LIN {X 0,Y 689.264,Z 377.17,A -85,B 0,C 180,E1 32346.673,E2 32346.673} C_VEL
LIN {X 0,Y 693.662,Z 395.744,A -85,B 0,C 180,E1 32346.172,E2 32346.172} C_VEL
LIN {X 0,Y 691.445,Z 657.884,A -85,B 0,C 180,E1 32343.063,E2 32343.063} C_VEL
LIN {X 0,Y 690.51,Z 767.576,A -85,B 0,C 180,E1 32341.762,E2 32341.762} C_VEL
LIN {X 0,Y 689.952,Z 793.018,A -85,B 0,C 180,E1 32341.311,E2 32341.311} C_VEL
LIN {X 0,Y 689.325,Z 814.667,A -85,B 0,C 180,E1 32340.791,E2 32340.791} C_VEL
LIN {X 0,Y 688.609,Z 838.554,A -85,B 0,C 180,E1 32340.063,E2 32340.063} C_VEL
LIN {X 0,Y 687.794,Z 859.592,A -85,B 0,C 180,E1 32339.277,E2 32339.277} C_VEL
LIN {X 0,Y 686.919,Z 881.255,A -85,B 0,C 180,E1 32338.329,E2 32338.329} C_VEL
LIN {X 0,Y 685.951,Z 903.052,A -85,B 0,C 180,E1 32337.197,E2 32337.197} C_VEL
LIN {X 0,Y 685.057,Z 922.955,A -85,B 0,C 180,E1 32336.012,E2 32336.012} C_VEL
LIN {X 0,Y 684.091,Z 943.292,A -85,B 0,C 180,E1 32334.613,E2 32334.613} C_VEL
LIN {X 0,Y 683.28,Z 961.609,A -85,B 0,C 180,E1 32333.182,E2 32333.182} C_VEL
LIN {X 0,Y 682.482,Z 979.534,A -85,B 0,C 180,E1 32331.576,E2 32331.576} C_VEL
LIN {X 0,Y 681.841,Z 995.625,A -85,B 0,C 180,E1 32329.948,E2 32329.948} C_VEL
LIN {X 0,Y 681.258,Z 1011.229,A -85,B 0,C 180,E1 32328.129,E2 32328.129} C_VEL
LIN {X 0,Y 680.802,Z 1025.061,A -85,B 0,C 180,E1 32326.291,E2 32326.291} C_VEL
LIN {X 0,Y 680.459,Z 1037.321,A -85,B 0,C 180,E1 32324.379,E2 32324.379} C_VEL
LIN {X 0,Y 680.233,Z 1047.861,A -85,B 0,C 180,E1 32322.479,E2 32322.479} C_VEL
LIN {X 0,Y 680.077,Z 1056.896,A -85,B 0,C 180,E1 32320.504,E2 32320.504} C_VEL
LIN {X 0,Y 679.969,Z 1063.726,A -85,B 0,C 180,E1 32318.712,E2 32318.712} C_VEL
LIN {X 0,Y 679.919,Z 1070.07,A -85,B 0,C 180,E1 32316.587,E2 32316.587} C_VEL
LIN {X 0,Y 679.921,Z 1073.974,A -85,B 0,C 180,E1 32314.808,E2 32314.808} C_VEL
LIN {X 0,Y 679.908,Z 1077.017,A -85,B 0,C 180,E1 32312.782,E2 32312.782} C_VEL
LIN {X 0,Y 679.899,Z 1078.306,A -85,B 0,C 180,E1 32310.758,E2 32310.758} C_VEL
LIN {X 0,Y 679.914,Z 1078.238,A -85,B 0,C 180,E1 32308.989,E2 32308.989} C_VEL
LIN {X 0,Y 679.916,Z 1076.461,A -85,B 0,C 180,E1 32306.796,E2 32306.796} C_VEL
LIN {X 0,Y 679.923,Z 1073.496,A -85,B 0,C 180,E1 32304.938,E2 32304.938} C_VEL
LIN {X 0,Y 679.954,Z 1068.507,A -85,B 0,C 180,E1 32302.82,E2 32302.82} C_VEL
LIN {X 0,Y 679.992,Z 1062.513,A -85,B 0,C 180,E1 32300.948,E2 32300.948} C_VEL
LIN {X 0,Y 680.097,Z 1055.12,A -85,B 0,C 180,E1 32299.067,E2 32299.067} C_VEL
LIN {X 0,Y 680.283,Z 1045.255,A -85,B 0,C 180,E1 32297.031,E2 32297.031} C_VEL
LIN {X 0,Y 680.52,Z 1035.245,A -85,B 0,C 180,E1 32295.274,E2 32295.274} C_VEL
LIN {X 0,Y 680.898,Z 1021.894,A -85,B 0,C 180,E1 32293.272,E2 32293.272} C_VEL
LIN {X 0,Y 681.318,Z 1009.107,A -85,B 0,C 180,E1 32291.607,E2 32291.607} C_VEL
LIN {X 0,Y 681.951,Z 992.791,A -85,B 0,C 180,E1 32289.755,E2 32289.755} C_VEL
LIN {X 0,Y 682.561,Z 977.636,A -85,B 0,C 180,E1 32288.242,E2 32288.242} C_VEL
LIN {X 0,Y 683.397,Z 958.847,A -85,B 0,C 180,E1 32286.595,E2 32286.595} C_VEL
LIN {X 0,Y 684.206,Z 940.792,A -85,B 0,C 180,E1 32285.202,E2 32285.202} C_VEL
LIN {X 0,Y 685.184,Z 919.997,A -85,B 0,C 180,E1 32283.804,E2 32283.804} C_VEL
LIN {X 0,Y 686.049,Z 900.695,A -85,B 0,C 180,E1 32282.671,E2 32282.671} C_VEL
LIN {X 0,Y 687.089,Z 877.282,A -85,B 0,C 180,E1 32281.489,E2 32281.489} C_VEL
LIN {X 0,Y 687.891,Z 857.092,A -85,B 0,C 180,E1 32280.622,E2 32280.622} C_VEL
LIN {X 0,Y 688.774,Z 832.985,A -85,B 0,C 180,E1 32279.752,E2 32279.752} C_VEL
LIN {X 0,Y 689.455,Z 811.007,A -85,B 0,C 180,E1 32279.114,E2 32279.114} C_VEL
LIN {X 0,Y 690.143,Z 786.732,A -85,B 0,C 180,E1 32278.559,E2 32278.559} C_VEL
LIN {X 0,Y 690.547,Z 763.43,A -85,B 0,C 180,E1 32278.181,E2 32278.181} C_VEL
LIN {X 0,Y 692.558,Z 519.957,A -85,B 0,C 180,E1 32275.31,E2 32275.31} C_VEL
LIN {X 0,Y 693.501,Z 394.27,A -85,B 0,C 180,E1 32273.8,E2 32273.8} C_VEL
LIN {X 0,Y 689.198,Z 376.448,A -85,B 0,C 180,E1 32273.293,E2 32273.293} C_VEL
LIN {X 0,Y 689.442,Z 360.316,A -85,B 0,C 180,E1 32272.089,E2 32272.089} C_VEL
LIN {X 0,Y 682.414,Z 342.087,A -85,B 0,C 180,E1 32270.221,E2 32270.221} C_VEL
LIN {X 0,Y 680.484,Z 336.477,A -85,B 0,C 180,E1 32269.637,E2 32269.637} C_VEL
LIN {X 0,Y 680.477,Z 336.471,A -85,B 0,C 180,E1 32266.543,E2 32266.543} C_VEL
LIN {X 0,Y 680.457,Z 336.467,A -85,B 0,C 180,E1 32263.914,E2 32263.914} C_VEL
LIN {X 0,Y 680.531,Z 336.466,A -85,B 0,C 180,E1 32260.943,E2 32260.943} C_VEL
LIN {X 0,Y 680.456,Z 336.464,A -85,B 0,C 180,E1 32258.036,E2 32258.036} C_VEL
LIN {X 0,Y 680.505,Z 336.462,A -85,B 0,C 180,E1 32255.219,E2 32255.219} C_VEL
LIN {X 0,Y 680.464,Z 336.464,A -85,B 0,C 180,E1 32252.136,E2 32252.136} C_VEL
LIN {X 0,Y 680.466,Z 336.462,A -85,B 0,C 180,E1 32249.489,E2 32249.489} C_VEL
LIN {X 0,Y 680.505,Z 336.463,A -85,B 0,C 180,E1 32246.437,E2 32246.437} C_VEL
LIN {X 0,Y 680.455,Z 336.457,A -85,B 0,C 180,E1 32243.651,E2 32243.651} C_VEL
LIN {X 0,Y 680.524,Z 336.46,A -85,B 0,C 180,E1 32240.828,E2 32240.828} C_VEL
LIN {X 0,Y 680.464,Z 336.464,A -85,B 0,C 180,E1 32237.885,E2 32237.885} C_VEL
LIN {X 0,Y 680.467,Z 336.46,A -85,B 0,C 180,E1 32235.25,E2 32235.25} C_VEL
LIN {X 0,Y 680.508,Z 336.467,A -85,B 0,C 180,E1 32232.215,E2 32232.215} C_VEL
LIN {X 0,Y 680.457,Z 336.454,A -85,B 0,C 180,E1 32229.387,E2 32229.387} C_VEL
LIN {X 0,Y 680.531,Z 336.461,A -85,B 0,C 180,E1 32226.496,E2 32226.496} C_VEL
LIN {X 0,Y 680.46,Z 336.462,A -85,B 0,C 180,E1 32223.538,E2 32223.538} C_VEL
LIN {X 0,Y 680.482,Z 336.461,A -85,B 0,C 180,E1 32220.842,E2 32220.842} C_VEL
LIN {X 0,Y 680.477,Z 336.466,A -85,B 0,C 180,E1 32217.691,E2 32217.691} C_VEL
LIN {X 0,Y 680.461,Z 336.459,A -85,B 0,C 180,E1 32215.026,E2 32215.026} C_VEL
LIN {X 0,Y 680.525,Z 336.463,A -85,B 0,C 180,E1 32212.014,E2 32212.014} C_VEL
LIN {X 0,Y 680.457,Z 336.454,A -85,B 0,C 180,E1 32209.159,E2 32209.159} C_VEL
LIN {X 0,Y 680.516,Z 336.459,A -85,B 0,C 180,E1 32206.316,E2 32206.316} C_VEL
LIN {X 0,Y 680.47,Z 336.462,A -85,B 0,C 180,E1 32203.346,E2 32203.346} C_VEL
LIN {X 0,Y 680.473,Z 336.461,A -85,B 0,C 180,E1 32200.623,E2 32200.623} C_VEL
LIN {X 0,Y 680.501,Z 336.467,A -85,B 0,C 180,E1 32197.54,E2 32197.54} C_VEL
LIN {X 0,Y 680.458,Z 336.455,A -85,B 0,C 180,E1 32194.777,E2 32194.777} C_VEL
LIN {X 0,Y 680.532,Z 336.463,A -85,B 0,C 180,E1 32191.832,E2 32191.832} C_VEL
LIN {X 0,Y 680.52,Z 336.461,A -85,B 0,C 180,E1 32189.539,E2 32189.539} C_VEL
LIN {X 0,Y 679.466,Z 336.601,A -85,B 0,C 180,E1 32188.891,E2 32188.891} C_VEL
LIN {X 0,Y 673.041,Z 337.385,A -85,B 0,C 180,E1 32187.073,E2 32187.073} C_VEL
LIN {X 0,Y 672.523,Z 337.446,A -85,B 0,C 180,E1 32186.601,E2 32186.601} C_VEL
LIN {X 0,Y 672.587,Z 337.449,A -85,B 0,C 180,E1 32183.618,E2 32183.618} C_VEL
LIN {X 0,Y 672.523,Z 337.451,A -85,B 0,C 180,E1 32180.701,E2 32180.701} C_VEL
LIN {X 0,Y 672.573,Z 337.452,A -85,B 0,C 180,E1 32177.889,E2 32177.889} C_VEL
LIN {X 0,Y 672.529,Z 337.444,A -85,B 0,C 180,E1 32174.807,E2 32174.807} C_VEL
LIN {X 0,Y 672.538,Z 337.449,A -85,B 0,C 180,E1 32172.107,E2 32172.107} C_VEL
LIN {X 0,Y 672.553,Z 337.459,A -85,B 0,C 180,E1 32168.963,E2 32168.963} C_VEL
LIN {X 0,Y 672.551,Z 337.617,A -85,B 0,C 180,E1 32166.62,E2 32166.62} C_VEL
LIN {X 0,Y 676.581,Z 348.492,A -85,B 0,C 180,E1 32165.427,E2 32165.427} C_VEL
LIN {X 0,Y 686.819,Z 366.483,A -85,B 0,C 180,E1 32164.54,E2 32164.54} C_VEL
LIN {X 0,Y 687.145,Z 369.523,A -85,B 0,C 180,E1 32164.481,E2 32164.481} C_VEL
LIN {X 0,Y 684.937,Z 605.975,A -85,B 0,C 180,E1 32161.643,E2 32161.643} C_VEL
LIN {X 0,Y 683.701,Z 737.454,A -85,B 0,C 180,E1 32160.073,E2 32160.073} C_VEL
LIN {X 0,Y 683.098,Z 762.982,A -85,B 0,C 180,E1 32159.617,E2 32159.617} C_VEL
LIN {X 0,Y 682.418,Z 784.428,A -85,B 0,C 180,E1 32159.099,E2 32159.099} C_VEL
LIN {X 0,Y 681.594,Z 808.728,A -85,B 0,C 180,E1 32158.353,E2 32158.353} C_VEL
LIN {X 0,Y 680.746,Z 828.609,A -85,B 0,C 180,E1 32157.607,E2 32157.607} C_VEL
LIN {X 0,Y 679.837,Z 849.314,A -85,B 0,C 180,E1 32156.7,E2 32156.7} C_VEL
LIN {X 0,Y 678.703,Z 872.036,A -85,B 0,C 180,E1 32155.526,E2 32155.526} C_VEL
LIN {X 0,Y 677.739,Z 891.66,A -85,B 0,C 180,E1 32154.353,E2 32154.353} C_VEL
LIN {X 0,Y 676.632,Z 912.524,A -85,B 0,C 180,E1 32152.916,E2 32152.916} C_VEL
LIN {X 0,Y 675.764,Z 930.2,A -85,B 0,C 180,E1 32151.528,E2 32151.528} C_VEL
LIN {X 0,Y 674.826,Z 949.063,A -85,B 0,C 180,E1 32149.835,E2 32149.835} C_VEL
LIN {X 0,Y 674.128,Z 964.72,A -85,B 0,C 180,E1 32148.238,E2 32148.238} C_VEL
LIN {X 0,Y 673.443,Z 980.568,A -85,B 0,C 180,E1 32146.386,E2 32146.386} C_VEL
LIN {X 0,Y 672.97,Z 993.715,A -85,B 0,C 180,E1 32144.63,E2 32144.63} C_VEL
LIN {X 0,Y 672.58,Z 1006.12,A -85,B 0,C 180,E1 32142.71,E2 32142.71} C_VEL
LIN {X 0,Y 672.312,Z 1015.81,A -85,B 0,C 180,E1 32140.974,E2 32140.974} C_VEL
LIN {X 0,Y 672.106,Z 1025.606,A -85,B 0,C 180,E1 32138.901,E2 32138.901} C_VEL
LIN {X 0,Y 672.002,Z 1032.768,A -85,B 0,C 180,E1 32137.043,E2 32137.043} C_VEL
LIN {X 0,Y 671.953,Z 1039.052,A -85,B 0,C 180,E1 32135.037,E2 32135.037} C_VEL
LIN {X 0,Y 671.917,Z 1043.668,A -85,B 0,C 180,E1 32132.986,E2 32132.986} C_VEL
LIN {X 0,Y 671.912,Z 1046.577,A -85,B 0,C 180,E1 32131.108,E2 32131.108} C_VEL
LIN {X 0,Y 671.911,Z 1048.239,A -85,B 0,C 180,E1 32128.977,E2 32128.977} C_VEL
LIN {X 0,Y 671.901,Z 1048.306,A -85,B 0,C 180,E1 32127.185,E2 32127.185} C_VEL
LIN {X 0,Y 671.901,Z 1047.011,A -85,B 0,C 180,E1 32125.134,E2 32125.134} C_VEL
LIN {X 0,Y 671.913,Z 1044.111,A -85,B 0,C 180,E1 32123.163,E2 32123.163} C_VEL
LIN {X 0,Y 671.93,Z 1040.23,A -85,B 0,C 180,E1 32121.356,E2 32121.356} C_VEL
LIN {X 0,Y 671.979,Z 1033.919,A -85,B 0,C 180,E1 32119.194,E2 32119.194} C_VEL
LIN {X 0,Y 672.093,Z 1027.074,A -85,B 0,C 180,E1 32117.368,E2 32117.368} C_VEL
LIN {X 0,Y 672.28,Z 1018.007,A -85,B 0,C 180,E1 32115.354,E2 32115.354} C_VEL
LIN {X 0,Y 672.542,Z 1007.386,A -85,B 0,C 180,E1 32113.414,E2 32113.414} C_VEL
LIN {X 0,Y 672.926,Z 995.003,A -85,B 0,C 180,E1 32111.459,E2 32111.459} C_VEL
LIN {X 0,Y 673.43,Z 980.998,A -85,B 0,C 180,E1 32109.579,E2 32109.579} C_VEL
LIN {X 0,Y 674.098,Z 965.519,A -85,B 0,C 180,E1 32107.757,E2 32107.757} C_VEL
LIN {X 0,Y 674.815,Z 949.282,A -85,B 0,C 180,E1 32106.097,E2 32106.097} C_VEL
LIN {X 0,Y 675.726,Z 930.994,A -85,B 0,C 180,E1 32104.447,E2 32104.447} C_VEL
LIN {X 0,Y 676.583,Z 913.495,A -85,B 0,C 180,E1 32103.066,E2 32103.066} C_VEL
LIN {X 0,Y 677.683,Z 892.893,A -85,B 0,C 180,E1 32101.634,E2 32101.634} C_VEL
LIN {X 0,Y 678.634,Z 873.594,A -85,B 0,C 180,E1 32100.472,E2 32100.472} C_VEL
LIN {X 0,Y 679.741,Z 851.422,A -85,B 0,C 180,E1 32099.307,E2 32099.307} C_VEL
LIN {X 0,Y 680.676,Z 830.276,A -85,B 0,C 180,E1 32098.371,E2 32098.371} C_VEL
LIN {X 0,Y 681.516,Z 810.536,A -85,B 0,C 180,E1 32097.621,E2 32097.621} C_VEL
LIN {X 0,Y 682.396,Z 785.089,A -85,B 0,C 180,E1 32096.829,E2 32096.829} C_VEL
LIN {X 0,Y 683.074,Z 763.638,A -85,B 0,C 180,E1 32096.307,E2 32096.307} C_VEL
LIN {X 0,Y 683.695,Z 738.242,A -85,B 0,C 180,E1 32095.848,E2 32095.848} C_VEL
LIN {X 0,Y 684.492,Z 656.332,A -85,B 0,C 180,E1 32094.862,E2 32094.862} C_VEL
LIN {X 0,Y 686.784,Z 406.301,A -85,B 0,C 180,E1 32091.875,E2 32091.875} C_VEL
LIN {X 0,Y 686.991,Z 367.172,A -85,B 0,C 180,E1 32091.39,E2 32091.39} C_VEL
LIN {X 0,Y 685.188,Z 363.29,A -85,B 0,C 180,E1 32091.227,E2 32091.227} C_VEL
LIN {X 0,Y 676.327,Z 347.874,A -85,B 0,C 180,E1 32090.437,E2 32090.437} C_VEL
LIN {X 0,Y 672.529,Z 337.459,A -85,B 0,C 180,E1 32089.255,E2 32089.255} C_VEL
LIN {X 0,Y 672.582,Z 337.45,A -85,B 0,C 180,E1 32086.262,E2 32086.262} C_VEL
LIN {X 0,Y 672.521,Z 337.451,A -85,B 0,C 180,E1 32083.362,E2 32083.362} C_VEL
LIN {X 0,Y 672.589,Z 337.433,A -85,B 0,C 180,E1 32080.404,E2 32080.404} C_VEL
LIN {X 0,Y 672.522,Z 337.452,A -85,B 0,C 180,E1 32077.445,E2 32077.445} C_VEL
LIN {X 0,Y 672.565,Z 337.438,A -85,B 0,C 180,E1 32074.605,E2 32074.605} C_VEL
LIN {X 0,Y 672.531,Z 337.446,A -85,B 0,C 180,E1 32071.557,E2 32071.557} C_VEL
LIN {X 0,Y 672.53,Z 337.454,A -85,B 0,C 180,E1 32068.872,E2 32068.872} C_VEL
LIN {X 0,Y 672.568,Z 337.445,A -85,B 0,C 180,E1 32065.823,E2 32065.823} C_VEL
LIN {X 0,Y 672.52,Z 337.454,A -85,B 0,C 180,E1 32063.018,E2 32063.018} C_VEL
LIN {X 0,Y 672.592,Z 337.453,A -85,B 0,C 180,E1 32060.085,E2 32060.085} C_VEL
LIN {X 0,Y 672.52,Z 337.449,A -85,B 0,C 180,E1 32057.121,E2 32057.121} C_VEL
LIN {X 0,Y 672.551,Z 337.453,A -85,B 0,C 180,E1 32054.376,E2 32054.376} C_VEL
LIN {X 0,Y 672.532,Z 337.45,A -85,B 0,C 180,E1 32051.231,E2 32051.231} C_VEL
LIN {X 0,Y 672.528,Z 337.451,A -85,B 0,C 180,E1 32048.55,E2 32048.55} C_VEL
LIN {X 0,Y 672.576,Z 337.446,A -85,B 0,C 180,E1 32045.545,E2 32045.545} C_VEL
LIN {X 0,Y 672.517,Z 337.453,A -85,B 0,C 180,E1 32042.727,E2 32042.727} C_VEL
LIN {X 0,Y 672.59,Z 337.453,A -85,B 0,C 180,E1 32039.83,E2 32039.83} C_VEL
LIN {X 0,Y 672.522,Z 337.445,A -85,B 0,C 180,E1 32036.847,E2 32036.847} C_VEL
LIN {X 0,Y 672.542,Z 337.456,A -85,B 0,C 180,E1 32034.112,E2 32034.112} C_VEL
LIN {X 0,Y 672.534,Z 337.451,A -85,B 0,C 180,E1 32030.933,E2 32030.933} C_VEL
LIN {X 0,Y 672.522,Z 337.446,A -85,B 0,C 180,E1 32028.247,E2 32028.247} C_VEL
LIN {X 0,Y 672.586,Z 337.441,A -85,B 0,C 180,E1 32025.273,E2 32025.273} C_VEL
LIN {X 0,Y 672.517,Z 337.453,A -85,B 0,C 180,E1 32022.37,E2 32022.37} C_VEL
LIN {X 0,Y 672.585,Z 337.45,A -85,B 0,C 180,E1 32019.461,E2 32019.461} C_VEL
LIN {X 0,Y 672.521,Z 337.445,A -85,B 0,C 180,E1 32016.518,E2 32016.518} C_VEL
LIN {X 0,Y 672.539,Z 337.455,A -85,B 0,C 180,E1 32013.796,E2 32013.796} C_VEL
LIN {X 0,Y 672.535,Z 337.45,A -85,B 0,C 180,E1 32010.602,E2 32010.602} C_VEL
LIN {X 0,Y 672.521,Z 337.455,A -85,B 0,C 180,E1 32007.937,E2 32007.937} C_VEL
LIN {X 0,Y 672.584,Z 337.452,A -85,B 0,C 180,E1 32004.981,E2 32004.981} C_VEL
LIN {X 0,Y 672.517,Z 337.453,A -85,B 0,C 180,E1 32002.117,E2 32002.117} C_VEL
LIN {X 0,Y 672.567,Z 337.455,A -85,B 0,C 180,E1 31999.306,E2 31999.306} C_VEL
LIN {X 0,Y 672.526,Z 337.453,A -85,B 0,C 180,E1 31996.263,E2 31996.263} C_VEL
LIN {X 0,Y 672.526,Z 337.458,A -85,B 0,C 180,E1 31993.609,E2 31993.609} C_VEL
LIN {X 0,Y 672.592,Z 337.467,A -85,B 0,C 180,E1 31990.826,E2 31990.826} C_VEL
LIN {X 0,Y 682.601,Z 364.163,A -85,B 0,C 180,E1 31988.045,E2 31988.045} C_VEL
LIN {X 0,Y 682.307,Z 376.941,A -85,B 0,C 180,E1 31987.109,E2 31987.109} C_VEL
LIN {X 0,Y 687.167,Z 397.582,A -85,B 0,C 180,E1 31986.542,E2 31986.542} C_VEL
LIN {X 0,Y 684.716,Z 660.338,A -85,B 0,C 180,E1 31983.4,E2 31983.4} C_VEL
LIN {X 0,Y 683.699,Z 767.71,A -85,B 0,C 180,E1 31982.114,E2 31982.114} C_VEL
LIN {X 0,Y 683.091,Z 793.146,A -85,B 0,C 180,E1 31981.658,E2 31981.658} C_VEL
LIN {X 0,Y 682.412,Z 814.556,A -85,B 0,C 180,E1 31981.14,E2 31981.14} C_VEL
LIN {X 0,Y 681.585,Z 838.968,A -85,B 0,C 180,E1 31980.39,E2 31980.39} C_VEL
LIN {X 0,Y 680.717,Z 859.347,A -85,B 0,C 180,E1 31979.622,E2 31979.622} C_VEL
LIN {X 0,Y 679.794,Z 880.266,A -85,B 0,C 180,E1 31978.701,E2 31978.701} C_VEL
LIN {X 0,Y 678.692,Z 902.317,A -85,B 0,C 180,E1 31977.555,E2 31977.555} C_VEL
LIN {X 0,Y 677.757,Z 921.216,A -85,B 0,C 180,E1 31976.426,E2 31976.426} C_VEL
LIN {X 0,Y 676.663,Z 942.008,A -85,B 0,C 180,E1 31975,E2 31975} C_VEL
LIN {X 0,Y 675.802,Z 959.4,A -85,B 0,C 180,E1 31973.638,E2 31973.638} C_VEL
LIN {X 0,Y 674.844,Z 978.606,A -85,B 0,C 180,E1 31971.924,E2 31971.924} C_VEL
LIN {X 0,Y 674.17,Z 993.722,A -85,B 0,C 180,E1 31970.389,E2 31970.389} C_VEL
LIN {X 0,Y 673.468,Z 1009.816,A -85,B 0,C 180,E1 31968.525,E2 31968.525} C_VEL
LIN {X 0,Y 673.008,Z 1022.525,A -85,B 0,C 180,E1 31966.841,E2 31966.841} C_VEL
LIN {X 0,Y 672.584,Z 1035.764,A -85,B 0,C 180,E1 31964.815,E2 31964.815} C_VEL
LIN {X 0,Y 672.325,Z 1045.586,A -85,B 0,C 180,E1 31963.061,E2 31963.061} C_VEL
LIN {X 0,Y 672.117,Z 1055.476,A -85,B 0,C 180,E1 31960.977,E2 31960.977} C_VEL
LIN {X 0,Y 672.012,Z 1062.514,A -85,B 0,C 180,E1 31959.161,E2 31959.161} C_VEL
LIN {X 0,Y 671.958,Z 1068.761,A -85,B 0,C 180,E1 31957.18,E2 31957.18} C_VEL
LIN {X 0,Y 671.924,Z 1073.497,A -85,B 0,C 180,E1 31955.123,E2 31955.123} C_VEL
LIN {X 0,Y 671.916,Z 1076.462,A -85,B 0,C 180,E1 31953.242,E2 31953.242} C_VEL
LIN {X 0,Y 671.914,Z 1078.238,A -85,B 0,C 180,E1 31951.023,E2 31951.023} C_VEL
LIN {X 0,Y 671.899,Z 1078.306,A -85,B 0,C 180,E1 31949.233,E2 31949.233} C_VEL
LIN {X 0,Y 671.909,Z 1077.017,A -85,B 0,C 180,E1 31947.185,E2 31947.185} C_VEL
LIN {X 0,Y 671.922,Z 1073.974,A -85,B 0,C 180,E1 31945.134,E2 31945.134} C_VEL
LIN {X 0,Y 671.923,Z 1070.07,A -85,B 0,C 180,E1 31943.335,E2 31943.335} C_VEL
LIN {X 0,Y 671.979,Z 1063.726,A -85,B 0,C 180,E1 31941.184,E2 31941.184} C_VEL
LIN {X 0,Y 672.097,Z 1056.896,A -85,B 0,C 180,E1 31939.369,E2 31939.369} C_VEL
LIN {X 0,Y 672.282,Z 1047.686,A -85,B 0,C 180,E1 31937.338,E2 31937.338} C_VEL
LIN {X 0,Y 672.539,Z 1037.261,A -85,B 0,C 180,E1 31935.437,E2 31935.437} C_VEL
LIN {X 0,Y 672.919,Z 1025.063,A -85,B 0,C 180,E1 31933.512,E2 31933.512} C_VEL
LIN {X 0,Y 673.423,Z 1011.227,A -85,B 0,C 180,E1 31931.653,E2 31931.653} C_VEL
LIN {X 0,Y 674.071,Z 996.17,A -85,B 0,C 180,E1 31929.871,E2 31929.871} C_VEL
LIN {X 0,Y 674.76,Z 980.459,A -85,B 0,C 180,E1 31928.256,E2 31928.256} C_VEL
LIN {X 0,Y 675.65,Z 962.715,A -85,B 0,C 180,E1 31926.634,E2 31926.634} C_VEL
LIN {X 0,Y 676.557,Z 944.067,A -85,B 0,C 180,E1 31925.154,E2 31925.154} C_VEL
LIN {X 0,Y 677.598,Z 924.668,A -85,B 0,C 180,E1 31923.792,E2 31923.792} C_VEL
LIN {X 0,Y 678.618,Z 903.936,A -85,B 0,C 180,E1 31922.537,E2 31922.537} C_VEL
LIN {X 0,Y 679.681,Z 882.64,A -85,B 0,C 180,E1 31921.41,E2 31921.41} C_VEL
LIN {X 0,Y 680.68,Z 860.265,A -85,B 0,C 180,E1 31920.415,E2 31920.415} C_VEL
LIN {X 0,Y 681.547,Z 839.834,A -85,B 0,C 180,E1 31919.641,E2 31919.641} C_VEL
LIN {X 0,Y 682.405,Z 814.776,A -85,B 0,C 180,E1 31918.866,E2 31918.866} C_VEL
LIN {X 0,Y 683.086,Z 793.282,A -85,B 0,C 180,E1 31918.344,E2 31918.344} C_VEL
LIN {X 0,Y 683.699,Z 767.822,A -85,B 0,C 180,E1 31917.887,E2 31917.887} C_VEL
LIN {X 0,Y 684.658,Z 666.935,A -85,B 0,C 180,E1 31916.678,E2 31916.678} C_VEL
LIN {X 0,Y 687.132,Z 401.239,A -85,B 0,C 180,E1 31913.502,E2 31913.502} C_VEL
LIN {X 0,Y 686.935,Z 395.795,A -85,B 0,C 180,E1 31913.42,E2 31913.42} C_VEL
LIN {X 0,Y 682.24,Z 376.221,A -85,B 0,C 180,E1 31912.856,E2 31912.856} C_VEL
LIN {X 0,Y 682.47,Z 363.779,A -85,B 0,C 180,E1 31911.917,E2 31911.917} C_VEL
LIN {X 0,Y 674.923,Z 343.947,A -85,B 0,C 180,E1 31909.858,E2 31909.858} C_VEL
LIN {X 0,Y 672.591,Z 337.458,A -85,B 0,C 180,E1 31909.148,E2 31909.148} C_VEL
LIN {X 0,Y 672.521,Z 337.459,A -85,B 0,C 180,E1 31906.263,E2 31906.263} C_VEL
LIN {X 0,Y 672.537,Z 337.455,A -85,B 0,C 180,E1 31903.611,E2 31903.611} C_VEL
LIN {X 0,Y 672.535,Z 337.451,A -85,B 0,C 180,E1 31900.408,E2 31900.408} C_VEL
LIN {X 0,Y 672.521,Z 337.451,A -85,B 0,C 180,E1 31897.724,E2 31897.724} C_VEL
LIN {X 0,Y 672.58,Z 337.449,A -85,B 0,C 180,E1 31894.703,E2 31894.703} C_VEL
LIN {X 0,Y 672.515,Z 337.451,A -85,B 0,C 180,E1 31891.858,E2 31891.858} C_VEL
LIN {X 0,Y 672.574,Z 337.449,A -85,B 0,C 180,E1 31889.055,E2 31889.055} C_VEL
LIN {X 0,Y 672.526,Z 337.454,A -85,B 0,C 180,E1 31886.015,E2 31886.015} C_VEL
LIN {X 0,Y 672.535,Z 337.443,A -85,B 0,C 180,E1 31883.296,E2 31883.296} C_VEL
LIN {X 0,Y 672.538,Z 337.449,A -85,B 0,C 180,E1 31880.087,E2 31880.087} C_VEL
LIN {X 0,Y 672.525,Z 337.451,A -85,B 0,C 180,E1 31877.349,E2 31877.349} C_VEL
LIN {X 0,Y 672.574,Z 337.446,A -85,B 0,C 180,E1 31874.287,E2 31874.287} C_VEL
LIN {X 0,Y 672.518,Z 337.452,A -85,B 0,C 180,E1 31871.492,E2 31871.492} C_VEL
LIN {X 0,Y 672.582,Z 337.44,A -85,B 0,C 180,E1 31868.636,E2 31868.636} C_VEL
LIN {X 0,Y 672.525,Z 337.449,A -85,B 0,C 180,E1 31865.631,E2 31865.631} C_VEL
LIN {X 0,Y 672.541,Z 337.447,A -85,B 0,C 180,E1 31862.897,E2 31862.897} C_VEL
LIN {X 0,Y 672.538,Z 337.444,A -85,B 0,C 180,E1 31859.744,E2 31859.744} C_VEL
LIN {X 0,Y 672.525,Z 337.451,A -85,B 0,C 180,E1 31857.017,E2 31857.017} C_VEL
LIN {X 0,Y 672.583,Z 337.444,A -85,B 0,C 180,E1 31854.022,E2 31854.022} C_VEL
LIN {X 0,Y 672.519,Z 337.453,A -85,B 0,C 180,E1 31851.191,E2 31851.191} C_VEL
LIN {X 0,Y 672.576,Z 337.439,A -85,B 0,C 180,E1 31848.335,E2 31848.335} C_VEL
LIN {X 0,Y 672.529,Z 337.451,A -85,B 0,C 180,E1 31845.36,E2 31845.36} C_VEL
LIN {X 0,Y 672.537,Z 337.447,A -85,B 0,C 180,E1 31842.612,E2 31842.612} C_VEL
LIN {X 0,Y 672.546,Z 337.446,A -85,B 0,C 180,E1 31839.46,E2 31839.46} C_VEL
LIN {X 0,Y 672.527,Z 337.452,A -85,B 0,C 180,E1 31836.704,E2 31836.704} C_VEL
LIN {X 0,Y 672.585,Z 337.446,A -85,B 0,C 180,E1 31833.694,E2 31833.694} C_VEL
LIN {X 0,Y 672.522,Z 337.445,A -85,B 0,C 180,E1 31830.813,E2 31830.813} C_VEL
LIN {X 0,Y 672.585,Z 337.45,A -85,B 0,C 180,E1 31827.928,E2 31827.928} C_VEL
LIN {X 0,Y 672.523,Z 337.446,A -85,B 0,C 180,E1 31826.601,E2 31826.601} C_VEL
LIN {X 0,Y 671.558,Z 337.57,A -85,B 0,C 180,E1 31825.945,E2 31825.945} C_VEL
LIN {X 0,Y 665.187,Z 338.373,A -85,B 0,C 180,E1 31824.105,E2 31824.105} C_VEL
LIN {X 0,Y 664.648,Z 338.437,A -85,B 0,C 180,E1 31823.627,E2 31823.627} C_VEL
LIN {X 0,Y 664.585,Z 338.44,A -85,B 0,C 180,E1 31820.698,E2 31820.698} C_VEL
LIN {X 0,Y 664.638,Z 338.441,A -85,B 0,C 180,E1 31817.858,E2 31817.858} C_VEL
LIN {X 0,Y 664.596,Z 338.429,A -85,B 0,C 180,E1 31814.877,E2 31814.877} C_VEL
LIN {X 0,Y 664.598,Z 338.439,A -85,B 0,C 180,E1 31812.121,E2 31812.121} C_VEL
LIN {X 0,Y 664.611,Z 338.448,A -85,B 0,C 180,E1 31808.939,E2 31808.939} C_VEL
LIN {X 0,Y 664.652,Z 338.576,A -85,B 0,C 180,E1 31807.103,E2 31807.103} C_VEL
LIN {X 0,Y 668.468,Z 348.792,A -85,B 0,C 180,E1 31805.961,E2 31805.961} C_VEL
LIN {X 0,Y 680.723,Z 370.08,A -85,B 0,C 180,E1 31804.878,E2 31804.878} C_VEL
LIN {X 0,Y 678.272,Z 606.578,A -85,B 0,C 180,E1 31802.012,E2 31802.012} C_VEL
LIN {X 0,Y 676.917,Z 737.51,A -85,B 0,C 180,E1 31800.433,E2 31800.433} C_VEL
LIN {X 0,Y 676.265,Z 763.04,A -85,B 0,C 180,E1 31799.973,E2 31799.973} C_VEL
LIN {X 0,Y 675.538,Z 784.266,A -85,B 0,C 180,E1 31799.456,E2 31799.456} C_VEL
LIN {X 0,Y 674.669,Z 807.51,A -85,B 0,C 180,E1 31798.746,E2 31798.746} C_VEL
LIN {X 0,Y 673.656,Z 829.251,A -85,B 0,C 180,E1 31797.923,E2 31797.923} C_VEL
LIN {X 0,Y 672.621,Z 850.868,A -85,B 0,C 180,E1 31796.962,E2 31796.962} C_VEL
LIN {X 0,Y 671.416,Z 872.5,A -85,B 0,C 180,E1 31795.823,E2 31795.823} C_VEL
LIN {X 0,Y 670.363,Z 892.083,A -85,B 0,C 180,E1 31794.639,E2 31794.639} C_VEL
LIN {X 0,Y 669.153,Z 912.814,A -85,B 0,C 180,E1 31793.192,E2 31793.192} C_VEL
LIN {X 0,Y 668.189,Z 930.522,A -85,B 0,C 180,E1 31791.784,E2 31791.784} C_VEL
LIN {X 0,Y 667.206,Z 948.416,A -85,B 0,C 180,E1 31790.162,E2 31790.162} C_VEL
LIN {X 0,Y 666.442,Z 963.293,A -85,B 0,C 180,E1 31788.637,E2 31788.637} C_VEL
LIN {X 0,Y 665.641,Z 980.076,A -85,B 0,C 180,E1 31786.673,E2 31786.673} C_VEL
LIN {X 0,Y 665.148,Z 992.639,A -85,B 0,C 180,E1 31784.985,E2 31784.985} C_VEL
LIN {X 0,Y 664.658,Z 1006.176,A -85,B 0,C 180,E1 31782.881,E2 31782.881} C_VEL
LIN {X 0,Y 664.357,Z 1015.988,A -85,B 0,C 180,E1 31781.098,E2 31781.098} C_VEL
LIN {X 0,Y 664.129,Z 1025.709,A -85,B 0,C 180,E1 31779.008,E2 31779.008} C_VEL
LIN {X 0,Y 664.025,Z 1032.677,A -85,B 0,C 180,E1 31777.18,E2 31777.18} C_VEL
LIN {X 0,Y 663.955,Z 1038.873,A -85,B 0,C 180,E1 31775.184,E2 31775.184} C_VEL
LIN {X 0,Y 663.92,Z 1043.554,A -85,B 0,C 180,E1 31773.108,E2 31773.108} C_VEL
LIN {X 0,Y 663.911,Z 1046.385,A -85,B 0,C 180,E1 31771.294,E2 31771.294} C_VEL
LIN {X 0,Y 663.912,Z 1048.199,A -85,B 0,C 180,E1 31769.137,E2 31769.137} C_VEL
LIN {X 0,Y 663.899,Z 1048.322,A -85,B 0,C 180,E1 31767.238,E2 31767.238} C_VEL
LIN {X 0,Y 663.898,Z 1047.134,A -85,B 0,C 180,E1 31765.248,E2 31765.248} C_VEL
LIN {X 0,Y 663.913,Z 1044.224,A -85,B 0,C 180,E1 31763.167,E2 31763.167} C_VEL
LIN {X 0,Y 663.933,Z 1040.377,A -85,B 0,C 180,E1 31761.338,E2 31761.338} C_VEL
LIN {X 0,Y 663.986,Z 1034.441,A -85,B 0,C 180,E1 31759.238,E2 31759.238} C_VEL
LIN {X 0,Y 664.109,Z 1027.328,A -85,B 0,C 180,E1 31757.302,E2 31757.302} C_VEL
LIN {X 0,Y 664.305,Z 1018.729,A -85,B 0,C 180,E1 31755.353,E2 31755.353} C_VEL
LIN {X 0,Y 664.592,Z 1008.272,A -85,B 0,C 180,E1 31753.39,E2 31753.39} C_VEL
LIN {X 0,Y 664.959,Z 997.182,A -85,B 0,C 180,E1 31751.592,E2 31751.592} C_VEL
LIN {X 0,Y 665.538,Z 982.914,A -85,B 0,C 180,E1 31749.601,E2 31749.601} C_VEL
LIN {X 0,Y 666.139,Z 969.457,A -85,B 0,C 180,E1 31747.96,E2 31747.96} C_VEL
LIN {X 0,Y 667.005,Z 952.253,A -85,B 0,C 180,E1 31746.125,E2 31746.125} C_VEL
LIN {X 0,Y 667.84,Z 936.516,A -85,B 0,C 180,E1 31744.647,E2 31744.647} C_VEL
LIN {X 0,Y 668.968,Z 916.216,A -85,B 0,C 180,E1 31742.975,E2 31742.975} C_VEL
LIN {X 0,Y 670.033,Z 897.67,A -85,B 0,C 180,E1 31741.641,E2 31741.641} C_VEL
LIN {X 0,Y 671.267,Z 875.582,A -85,B 0,C 180,E1 31740.263,E2 31740.263} C_VEL
LIN {X 0,Y 672.336,Z 855.537,A -85,B 0,C 180,E1 31739.18,E2 31739.18} C_VEL
LIN {X 0,Y 673.539,Z 831.903,A -85,B 0,C 180,E1 31738.096,E2 31738.096} C_VEL
LIN {X 0,Y 674.443,Z 812.39,A -85,B 0,C 180,E1 31737.341,E2 31737.341} C_VEL
LIN {X 0,Y 675.396,Z 788.595,A -85,B 0,C 180,E1 31736.57,E2 31736.57} C_VEL
LIN {X 0,Y 676.156,Z 765.864,A -85,B 0,C 180,E1 31735.999,E2 31735.999} C_VEL
LIN {X 0,Y 676.874,Z 741.591,A -85,B 0,C 180,E1 31735.535,E2 31735.535} C_VEL
LIN {X 0,Y 677.412,Z 695.138,A -85,B 0,C 180,E1 31734.953,E2 31734.953} C_VEL
LIN {X 0,Y 679.97,Z 442.631,A -85,B 0,C 180,E1 31731.92,E2 31731.92} C_VEL
LIN {X 0,Y 680.612,Z 369.671,A -85,B 0,C 180,E1 31731.02,E2 31731.02} C_VEL
LIN {X 0,Y 668.308,Z 348.44,A -85,B 0,C 180,E1 31729.932,E2 31729.932} C_VEL
LIN {X 0,Y 664.639,Z 338.439,A -85,B 0,C 180,E1 31728.782,E2 31728.782} C_VEL
LIN {X 0,Y 664.589,Z 338.441,A -85,B 0,C 180,E1 31725.725,E2 31725.725} C_VEL
LIN {X 0,Y 664.604,Z 338.442,A -85,B 0,C 180,E1 31722.964,E2 31722.964} C_VEL
LIN {X 0,Y 664.597,Z 338.435,A -85,B 0,C 180,E1 31719.748,E2 31719.748} C_VEL
LIN {X 0,Y 664.593,Z 338.44,A -85,B 0,C 180,E1 31717,E2 31717} C_VEL
LIN {X 0,Y 664.619,Z 338.439,A -85,B 0,C 180,E1 31713.854,E2 31713.854} C_VEL
LIN {X 0,Y 664.585,Z 338.437,A -85,B 0,C 180,E1 31711.068,E2 31711.068} C_VEL
LIN {X 0,Y 664.653,Z 338.437,A -85,B 0,C 180,E1 31708.091,E2 31708.091} C_VEL
LIN {X 0,Y 664.58,Z 338.436,A -85,B 0,C 180,E1 31705.201,E2 31705.201} C_VEL
LIN {X 0,Y 664.631,Z 338.441,A -85,B 0,C 180,E1 31702.372,E2 31702.372} C_VEL
LIN {X 0,Y 664.592,Z 338.44,A -85,B 0,C 180,E1 31699.329,E2 31699.329} C_VEL
LIN {X 0,Y 664.597,Z 338.441,A -85,B 0,C 180,E1 31696.59,E2 31696.59} C_VEL
LIN {X 0,Y 664.604,Z 338.437,A -85,B 0,C 180,E1 31693.397,E2 31693.397} C_VEL
LIN {X 0,Y 664.584,Z 338.442,A -85,B 0,C 180,E1 31690.665,E2 31690.665} C_VEL
LIN {X 0,Y 664.645,Z 338.437,A -85,B 0,C 180,E1 31687.608,E2 31687.608} C_VEL
LIN {X 0,Y 664.579,Z 338.438,A -85,B 0,C 180,E1 31684.747,E2 31684.747} C_VEL
LIN {X 0,Y 664.647,Z 338.434,A -85,B 0,C 180,E1 31681.81,E2 31681.81} C_VEL
LIN {X 0,Y 664.585,Z 338.441,A -85,B 0,C 180,E1 31678.879,E2 31678.879} C_VEL
LIN {X 0,Y 664.606,Z 338.437,A -85,B 0,C 180,E1 31676.118,E2 31676.118} C_VEL
LIN {X 0,Y 664.596,Z 338.431,A -85,B 0,C 180,E1 31673,E2 31673} C_VEL
LIN {X 0,Y 664.584,Z 338.443,A -85,B 0,C 180,E1 31670.299,E2 31670.299} C_VEL
LIN {X 0,Y 664.636,Z 338.438,A -85,B 0,C 180,E1 31667.223,E2 31667.223} C_VEL
LIN {X 0,Y 664.578,Z 338.434,A -85,B 0,C 180,E1 31664.376,E2 31664.376} C_VEL
LIN {X 0,Y 664.651,Z 338.433,A -85,B 0,C 180,E1 31661.402,E2 31661.402} C_VEL
LIN {X 0,Y 664.58,Z 338.442,A -85,B 0,C 180,E1 31658.405,E2 31658.405} C_VEL
LIN {X 0,Y 664.631,Z 338.438,A -85,B 0,C 180,E1 31655.561,E2 31655.561} C_VEL
LIN {X 0,Y 664.587,Z 338.437,A -85,B 0,C 180,E1 31652.491,E2 31652.491} C_VEL
LIN {X 0,Y 664.591,Z 338.443,A -85,B 0,C 180,E1 31649.834,E2 31649.834} C_VEL
LIN {X 0,Y 664.613,Z 338.441,A -85,B 0,C 180,E1 31646.692,E2 31646.692} C_VEL
LIN {X 0,Y 664.58,Z 338.444,A -85,B 0,C 180,E1 31643.965,E2 31643.965} C_VEL
LIN {X 0,Y 664.653,Z 338.44,A -85,B 0,C 180,E1 31641.036,E2 31641.036} C_VEL
LIN {X 0,Y 664.579,Z 338.443,A -85,B 0,C 180,E1 31638.085,E2 31638.085} C_VEL
LIN {X 0,Y 664.627,Z 338.442,A -85,B 0,C 180,E1 31635.243,E2 31635.243} C_VEL
LIN {X 0,Y 664.585,Z 338.443,A -85,B 0,C 180,E1 31632.146,E2 31632.146} C_VEL
LIN {X 0,Y 664.621,Z 338.542,A -85,B 0,C 180,E1 31631.317,E2 31631.317} C_VEL
LIN {X 0,Y 673.506,Z 362.08,A -85,B 0,C 180,E1 31628.792,E2 31628.792} C_VEL
LIN {X 0,Y 675.561,Z 368.02,A -85,B 0,C 180,E1 31628.193,E2 31628.193} C_VEL
LIN {X 0,Y 675.363,Z 376.661,A -85,B 0,C 180,E1 31627.557,E2 31627.557} C_VEL
LIN {X 0,Y 680.703,Z 399.355,A -85,B 0,C 180,E1 31626.921,E2 31626.921} C_VEL
LIN {X 0,Y 678.008,Z 663.113,A -85,B 0,C 180,E1 31623.74,E2 31623.74} C_VEL
LIN {X 0,Y 676.914,Z 767.818,A -85,B 0,C 180,E1 31622.474,E2 31622.474} C_VEL
LIN {X 0,Y 676.255,Z 793.274,A -85,B 0,C 180,E1 31622.013,E2 31622.013} C_VEL
LIN {X 0,Y 675.528,Z 814.444,A -85,B 0,C 180,E1 31621.497,E2 31621.497} C_VEL
LIN {X 0,Y 674.622,Z 838.547,A -85,B 0,C 180,E1 31620.753,E2 31620.753} C_VEL
LIN {X 0,Y 673.655,Z 859.342,A -85,B 0,C 180,E1 31619.964,E2 31619.964} C_VEL
LIN {X 0,Y 672.656,Z 880.17,A -85,B 0,C 180,E1 31619.039,E2 31619.039} C_VEL
LIN {X 0,Y 671.429,Z 902.313,A -85,B 0,C 180,E1 31617.879,E2 31617.879} C_VEL
LIN {X 0,Y 670.354,Z 922.188,A -85,B 0,C 180,E1 31616.677,E2 31616.677} C_VEL
LIN {X 0,Y 669.167,Z 942.614,A -85,B 0,C 180,E1 31615.252,E2 31615.252} C_VEL
LIN {X 0,Y 668.229,Z 959.683,A -85,B 0,C 180,E1 31613.899,E2 31613.899} C_VEL
LIN {X 0,Y 667.192,Z 978.606,A -85,B 0,C 180,E1 31612.189,E2 31612.189} C_VEL
LIN {X 0,Y 666.433,Z 993.633,A -85,B 0,C 180,E1 31610.645,E2 31610.645} C_VEL
LIN {X 0,Y 665.654,Z 1009.818,A -85,B 0,C 180,E1 31608.751,E2 31608.751} C_VEL
LIN {X 0,Y 665.145,Z 1022.539,A -85,B 0,C 180,E1 31607.044,E2 31607.044} C_VEL
LIN {X 0,Y 664.665,Z 1035.765,A -85,B 0,C 180,E1 31604.996,E2 31604.996} C_VEL
LIN {X 0,Y 664.369,Z 1045.92,A -85,B 0,C 180,E1 31603.156,E2 31603.156} C_VEL
LIN {X 0,Y 664.133,Z 1055.927,A -85,B 0,C 180,E1 31601,E2 31601} C_VEL
LIN {X 0,Y 664.022,Z 1062.817,A -85,B 0,C 180,E1 31599.185,E2 31599.185} C_VEL
LIN {X 0,Y 663.962,Z 1069.244,A -85,B 0,C 180,E1 31597.093,E2 31597.093} C_VEL
LIN {X 0,Y 663.925,Z 1073.656,A -85,B 0,C 180,E1 31595.098,E2 31595.098} C_VEL
LIN {X 0,Y 663.917,Z 1076.574,A -85,B 0,C 180,E1 31593.194,E2 31593.194} C_VEL
LIN {X 0,Y 663.91,Z 1078.261,A -85,B 0,C 180,E1 31590.949,E2 31590.949} C_VEL
LIN {X 0,Y 663.905,Z 1078.283,A -85,B 0,C 180,E1 31589.137,E2 31589.137} C_VEL
LIN {X 0,Y 663.916,Z 1076.799,A -85,B 0,C 180,E1 31586.978,E2 31586.978} C_VEL
LIN {X 0,Y 663.925,Z 1073.815,A -85,B 0,C 180,E1 31584.989,E2 31584.989} C_VEL
LIN {X 0,Y 663.956,Z 1069.451,A -85,B 0,C 180,E1 31582.993,E2 31582.993} C_VEL
LIN {X 0,Y 664.011,Z 1063.119,A -85,B 0,C 180,E1 31580.903,E2 31580.903} C_VEL
LIN {X 0,Y 664.128,Z 1056.186,A -85,B 0,C 180,E1 31579.065,E2 31579.065} C_VEL
LIN {X 0,Y 664.356,Z 1046.484,A -85,B 0,C 180,E1 31576.953,E2 31576.953} C_VEL
LIN {X 0,Y 664.649,Z 1036.288,A -85,B 0,C 180,E1 31575.093,E2 31575.093} C_VEL
LIN {X 0,Y 665.121,Z 1023.16,A -85,B 0,C 180,E1 31573.044,E2 31573.044} C_VEL
LIN {X 0,Y 665.624,Z 1010.525,A -85,B 0,C 180,E1 31571.339,E2 31571.339} C_VEL
LIN {X 0,Y 666.404,Z 994.378,A -85,B 0,C 180,E1 31569.435,E2 31569.435} C_VEL
LIN {X 0,Y 667.168,Z 979.013,A -85,B 0,C 180,E1 31567.851,E2 31567.851} C_VEL
LIN {X 0,Y 668.189,Z 960.506,A -85,B 0,C 180,E1 31566.17,E2 31566.17} C_VEL
LIN {X 0,Y 669.129,Z 943.22,A -85,B 0,C 180,E1 31564.794,E2 31564.794} C_VEL
LIN {X 0,Y 670.317,Z 922.909,A -85,B 0,C 180,E1 31563.369,E2 31563.369} C_VEL
LIN {X 0,Y 671.389,Z 903.048,A -85,B 0,C 180,E1 31562.163,E2 31562.163} C_VEL
LIN {X 0,Y 672.604,Z 881.268,A -85,B 0,C 180,E1 31561.012,E2 31561.012} C_VEL
LIN {X 0,Y 673.605,Z 860.476,A -85,B 0,C 180,E1 31560.082,E2 31560.082} C_VEL
LIN {X 0,Y 674.538,Z 840.351,A -85,B 0,C 180,E1 31559.312,E2 31559.312} C_VEL
LIN {X 0,Y 675.503,Z 815.099,A -85,B 0,C 180,E1 31558.521,E2 31558.521} C_VEL
LIN {X 0,Y 676.235,Z 793.801,A -85,B 0,C 180,E1 31557.998,E2 31557.998} C_VEL
LIN {X 0,Y 676.909,Z 768.357,A -85,B 0,C 180,E1 31557.534,E2 31557.534} C_VEL
LIN {X 0,Y 677.778,Z 687.025,A -85,B 0,C 180,E1 31556.545,E2 31556.545} C_VEL
LIN {X 0,Y 680.316,Z 433.987,A -85,B 0,C 180,E1 31553.5,E2 31553.5} C_VEL
LIN {X 0,Y 680.519,Z 397.746,A -85,B 0,C 180,E1 31553.046,E2 31553.046} C_VEL
LIN {X 0,Y 675.309,Z 375.991,A -85,B 0,C 180,E1 31552.409,E2 31552.409} C_VEL
LIN {X 0,Y 675.511,Z 367.275,A -85,B 0,C 180,E1 31551.744,E2 31551.744} C_VEL
LIN {X 0,Y 667.62,Z 346.692,A -85,B 0,C 180,E1 31549.571,E2 31549.571} C_VEL
LIN {X 0,Y 664.607,Z 338.449,A -85,B 0,C 180,E1 31548.655,E2 31548.655} C_VEL
LIN {X 0,Y 664.579,Z 338.447,A -85,B 0,C 180,E1 31545.965,E2 31545.965} C_VEL
LIN {X 0,Y 664.647,Z 338.444,A -85,B 0,C 180,E1 31542.96,E2 31542.96} C_VEL
LIN {X 0,Y 664.579,Z 338.439,A -85,B 0,C 180,E1 31540.087,E2 31540.087} C_VEL
LIN {X 0,Y 664.618,Z 338.438,A -85,B 0,C 180,E1 31537.322,E2 31537.322} C_VEL
LIN {X 0,Y 664.591,Z 338.44,A -85,B 0,C 180,E1 31534.242,E2 31534.242} C_VEL
LIN {X 0,Y 664.585,Z 338.439,A -85,B 0,C 180,E1 31531.573,E2 31531.573} C_VEL
LIN {X 0,Y 664.636,Z 338.439,A -85,B 0,C 180,E1 31528.529,E2 31528.529} C_VEL
LIN {X 0,Y 664.579,Z 338.441,A -85,B 0,C 180,E1 31525.678,E2 31525.678} C_VEL
LIN {X 0,Y 664.652,Z 338.43,A -85,B 0,C 180,E1 31522.745,E2 31522.745} C_VEL
LIN {X 0,Y 664.581,Z 338.436,A -85,B 0,C 180,E1 31519.787,E2 31519.787} C_VEL
LIN {X 0,Y 664.62,Z 338.438,A -85,B 0,C 180,E1 31516.97,E2 31516.97} C_VEL
LIN {X 0,Y 664.595,Z 338.44,A -85,B 0,C 180,E1 31513.929,E2 31513.929} C_VEL
LIN {X 0,Y 664.589,Z 338.44,A -85,B 0,C 180,E1 31511.191,E2 31511.191} C_VEL
LIN {X 0,Y 664.617,Z 338.445,A -85,B 0,C 180,E1 31508.043,E2 31508.043} C_VEL
LIN {X 0,Y 664.581,Z 338.436,A -85,B 0,C 180,E1 31505.266,E2 31505.266} C_VEL
LIN {X 0,Y 664.649,Z 338.44,A -85,B 0,C 180,E1 31502.242,E2 31502.242} C_VEL
LIN {X 0,Y 664.58,Z 338.43,A -85,B 0,C 180,E1 31499.397,E2 31499.397} C_VEL
LIN {X 0,Y 664.629,Z 338.438,A -85,B 0,C 180,E1 31496.55,E2 31496.55} C_VEL
LIN {X 0,Y 664.592,Z 338.438,A -85,B 0,C 180,E1 31493.521,E2 31493.521} C_VEL
LIN {X 0,Y 664.593,Z 338.44,A -85,B 0,C 180,E1 31490.823,E2 31490.823} C_VEL
LIN {X 0,Y 664.615,Z 338.443,A -85,B 0,C 180,E1 31487.665,E2 31487.665} C_VEL
LIN {X 0,Y 664.584,Z 338.437,A -85,B 0,C 180,E1 31484.913,E2 31484.913} C_VEL
LIN {X 0,Y 664.65,Z 338.438,A -85,B 0,C 180,E1 31481.946,E2 31481.946} C_VEL
LIN {X 0,Y 664.582,Z 338.434,A -85,B 0,C 180,E1 31479.018,E2 31479.018} C_VEL
LIN {X 0,Y 664.64,Z 338.439,A -85,B 0,C 180,E1 31476.128,E2 31476.128} C_VEL
LIN {X 0,Y 664.589,Z 338.443,A -85,B 0,C 180,E1 31473.072,E2 31473.072} C_VEL
LIN {X 0,Y 664.605,Z 338.431,A -85,B 0,C 180,E1 31470.332,E2 31470.332} C_VEL
LIN {X 0,Y 664.605,Z 338.436,A -85,B 0,C 180,E1 31467.206,E2 31467.206} C_VEL
LIN {X 0,Y 664.589,Z 338.441,A -85,B 0,C 180,E1 31464.483,E2 31464.483} C_VEL
LIN {X 0,Y 664.648,Z 338.437,A -85,B 0,C 180,E1 31463.627,E2 31463.627} C_VEL
LIN {X 0,Y 663.642,Z 338.561,A -85,B 0,C 180,E1 31462.963,E2 31462.963} C_VEL
LIN {X 0,Y 657.183,Z 339.369,A -85,B 0,C 180,E1 31461.102,E2 31461.102} C_VEL
LIN {X 0,Y 656.644,Z 339.428,A -85,B 0,C 180,E1 31460.617,E2 31460.617} C_VEL
LIN {X 0,Y 656.711,Z 339.428,A -85,B 0,C 180,E1 31457.702,E2 31457.702} C_VEL
LIN {X 0,Y 656.647,Z 339.421,A -85,B 0,C 180,E1 31454.674,E2 31454.674} C_VEL
LIN {X 0,Y 656.688,Z 339.425,A -85,B 0,C 180,E1 31451.829,E2 31451.829} C_VEL
LIN {X 0,Y 656.656,Z 339.438,A -85,B 0,C 180,E1 31448.743,E2 31448.743} C_VEL
LIN {X 0,Y 656.715,Z 339.481,A -85,B 0,C 180,E1 31447.608,E2 31447.608} C_VEL
LIN {X 0,Y 660.299,Z 349.162,A -85,B 0,C 180,E1 31446.516,E2 31446.516} C_VEL
LIN {X 0,Y 672.665,Z 370.1,A -85,B 0,C 180,E1 31445.399,E2 31445.399} C_VEL
LIN {X 0,Y 674.3,Z 373.32,A -85,B 0,C 180,E1 31445.249,E2 31445.249} C_VEL
LIN {X 0,Y 671.62,Z 610.125,A -85,B 0,C 180,E1 31442.354,E2 31442.354} C_VEL
LIN {X 0,Y 670.159,Z 737.628,A -85,B 0,C 180,E1 31440.8,E2 31440.8} C_VEL
LIN {X 0,Y 669.456,Z 763.152,A -85,B 0,C 180,E1 31440.336,E2 31440.336} C_VEL
LIN {X 0,Y 668.682,Z 784.147,A -85,B 0,C 180,E1 31439.821,E2 31439.821} C_VEL
LIN {X 0,Y 667.747,Z 806.973,A -85,B 0,C 180,E1 31439.121,E2 31439.121} C_VEL
LIN {X 0,Y 666.641,Z 828.781,A -85,B 0,C 180,E1 31438.292,E2 31438.292} C_VEL
LIN {X 0,Y 665.571,Z 849.482,A -85,B 0,C 180,E1 31437.368,E2 31437.368} C_VEL
LIN {X 0,Y 664.202,Z 872.164,A -85,B 0,C 180,E1 31436.173,E2 31436.173} C_VEL
LIN {X 0,Y 663.039,Z 891.79,A -85,B 0,C 180,E1 31434.977,E2 31434.977} C_VEL
LIN {X 0,Y 661.729,Z 912.624,A -85,B 0,C 180,E1 31433.51,E2 31433.51} C_VEL
LIN {X 0,Y 660.649,Z 930.299,A -85,B 0,C 180,E1 31432.093,E2 31432.093} C_VEL
LIN {X 0,Y 659.548,Z 948.684,A -85,B 0,C 180,E1 31430.407,E2 31430.407} C_VEL
LIN {X 0,Y 658.704,Z 963.538,A -85,B 0,C 180,E1 31428.864,E2 31428.864} C_VEL
LIN {X 0,Y 657.869,Z 979.584,A -85,B 0,C 180,E1 31426.967,E2 31426.967} C_VEL
LIN {X 0,Y 657.3,Z 992.193,A -85,B 0,C 180,E1 31425.258,E2 31425.258} C_VEL
LIN {X 0,Y 656.765,Z 1005.394,A -85,B 0,C 180,E1 31423.201,E2 31423.201} C_VEL
LIN {X 0,Y 656.44,Z 1015.162,A -85,B 0,C 180,E1 31421.421,E2 31421.421} C_VEL
LIN {X 0,Y 656.198,Z 1024.753,A -85,B 0,C 180,E1 31419.384,E2 31419.384} C_VEL
LIN {X 0,Y 656.045,Z 1032.462,A -85,B 0,C 180,E1 31417.356,E2 31417.356} C_VEL
LIN {X 0,Y 655.954,Z 1038.693,A -85,B 0,C 180,E1 31415.335,E2 31415.335} C_VEL
LIN {X 0,Y 655.916,Z 1043.44,A -85,B 0,C 180,E1 31413.233,E2 31413.233} C_VEL
LIN {X 0,Y 655.912,Z 1046.306,A -85,B 0,C 180,E1 31411.398,E2 31411.398} C_VEL
LIN {X 0,Y 655.909,Z 1048.183,A -85,B 0,C 180,E1 31409.214,E2 31409.214} C_VEL
LIN {X 0,Y 655.896,Z 1048.337,A -85,B 0,C 180,E1 31407.291,E2 31407.291} C_VEL
LIN {X 0,Y 655.897,Z 1047.251,A -85,B 0,C 180,E1 31405.366,E2 31405.366} C_VEL
LIN {X 0,Y 655.914,Z 1044.339,A -85,B 0,C 180,E1 31403.171,E2 31403.171} C_VEL
LIN {X 0,Y 655.935,Z 1040.525,A -85,B 0,C 180,E1 31401.32,E2 31401.32} C_VEL
LIN {X 0,Y 655.991,Z 1034.958,A -85,B 0,C 180,E1 31399.283,E2 31399.283} C_VEL
LIN {X 0,Y 656.126,Z 1027.58,A -85,B 0,C 180,E1 31397.234,E2 31397.234} C_VEL
LIN {X 0,Y 656.332,Z 1019.332,A -85,B 0,C 180,E1 31395.329,E2 31395.329} C_VEL
LIN {X 0,Y 656.66,Z 1008.638,A -85,B 0,C 180,E1 31393.274,E2 31393.274} C_VEL
LIN {X 0,Y 657.063,Z 997.584,A -85,B 0,C 180,E1 31391.453,E2 31391.453} C_VEL
LIN {X 0,Y 657.693,Z 983.412,A -85,B 0,C 180,E1 31389.44,E2 31389.44} C_VEL
LIN {X 0,Y 658.362,Z 970.013,A -85,B 0,C 180,E1 31387.78,E2 31387.78} C_VEL
LIN {X 0,Y 659.305,Z 952.896,A -85,B 0,C 180,E1 31385.922,E2 31385.922} C_VEL
LIN {X 0,Y 660.218,Z 937.24,A -85,B 0,C 180,E1 31384.429,E2 31384.429} C_VEL
LIN {X 0,Y 661.416,Z 917.701,A -85,B 0,C 180,E1 31382.787,E2 31382.787} C_VEL
LIN {X 0,Y 662.557,Z 899.324,A -85,B 0,C 180,E1 31381.441,E2 31381.441} C_VEL
LIN {X 0,Y 663.909,Z 877.57,A -85,B 0,C 180,E1 31380.049,E2 31380.049} C_VEL
LIN {X 0,Y 665.051,Z 857.744,A -85,B 0,C 180,E1 31378.956,E2 31378.956} C_VEL
LIN {X 0,Y 666.366,Z 834.681,A -85,B 0,C 180,E1 31377.864,E2 31377.864} C_VEL
LIN {X 0,Y 667.387,Z 814.243,A -85,B 0,C 180,E1 31377.054,E2 31377.054} C_VEL
LIN {X 0,Y 668.356,Z 792.889,A -85,B 0,C 180,E1 31376.339,E2 31376.339} C_VEL
LIN {X 0,Y 669.253,Z 768.222,A -85,B 0,C 180,E1 31375.687,E2 31375.687} C_VEL
LIN {X 0,Y 669.946,Z 746.408,A -85,B 0,C 180,E1 31375.25,E2 31375.25} C_VEL
LIN {X 0,Y 670.503,Z 714.244,A -85,B 0,C 180,E1 31374.808,E2 31374.808} C_VEL
LIN {X 0,Y 673.317,Z 459.697,A -85,B 0,C 180,E1 31371.727,E2 31371.727} C_VEL
LIN {X 0,Y 674.117,Z 372.503,A -85,B 0,C 180,E1 31370.638,E2 31370.638} C_VEL
LIN {X 0,Y 662.206,Z 352.425,A -85,B 0,C 180,E1 31369.57,E2 31369.57} C_VEL
LIN {X 0,Y 659.951,Z 348.526,A -85,B 0,C 180,E1 31369.346,E2 31369.346} C_VEL
LIN {X 0,Y 656.699,Z 339.432,A -85,B 0,C 180,E1 31368.252,E2 31368.252} C_VEL
LIN {X 0,Y 656.644,Z 339.431,A -85,B 0,C 180,E1 31365.414,E2 31365.414} C_VEL
LIN {X 0,Y 656.713,Z 339.426,A -85,B 0,C 180,E1 31362.415,E2 31362.415} C_VEL
LIN {X 0,Y 656.644,Z 339.425,A -85,B 0,C 180,E1 31359.464,E2 31359.464} C_VEL
LIN {X 0,Y 656.686,Z 339.413,A -85,B 0,C 180,E1 31356.638,E2 31356.638} C_VEL
LIN {X 0,Y 656.653,Z 339.43,A -85,B 0,C 180,E1 31353.556,E2 31353.556} C_VEL
LIN {X 0,Y 656.662,Z 339.428,A -85,B 0,C 180,E1 31350.772,E2 31350.772} C_VEL
LIN {X 0,Y 656.661,Z 339.429,A -85,B 0,C 180,E1 31347.574,E2 31347.574} C_VEL
LIN {X 0,Y 656.65,Z 339.426,A -85,B 0,C 180,E1 31344.833,E2 31344.833} C_VEL
LIN {X 0,Y 656.688,Z 339.422,A -85,B 0,C 180,E1 31341.716,E2 31341.716} C_VEL
LIN {X 0,Y 656.643,Z 339.431,A -85,B 0,C 180,E1 31338.926,E2 31338.926} C_VEL
LIN {X 0,Y 656.712,Z 339.428,A -85,B 0,C 180,E1 31335.906,E2 31335.906} C_VEL
LIN {X 0,Y 656.642,Z 339.428,A -85,B 0,C 180,E1 31332.955,E2 31332.955} C_VEL
LIN {X 0,Y 656.706,Z 339.423,A -85,B 0,C 180,E1 31329.996,E2 31329.996} C_VEL
LIN {X 0,Y 656.646,Z 339.429,A -85,B 0,C 180,E1 31326.997,E2 31326.997} C_VEL
LIN {X 0,Y 656.675,Z 339.429,A -85,B 0,C 180,E1 31324.181,E2 31324.181} C_VEL
LIN {X 0,Y 656.652,Z 339.423,A -85,B 0,C 180,E1 31321.047,E2 31321.047} C_VEL
LIN {X 0,Y 656.651,Z 339.433,A -85,B 0,C 180,E1 31318.342,E2 31318.342} C_VEL
LIN {X 0,Y 656.676,Z 339.428,A -85,B 0,C 180,E1 31315.196,E2 31315.196} C_VEL
LIN {X 0,Y 656.642,Z 339.423,A -85,B 0,C 180,E1 31312.387,E2 31312.387} C_VEL
LIN {X 0,Y 656.706,Z 339.419,A -85,B 0,C 180,E1 31309.384,E2 31309.384} C_VEL
LIN {X 0,Y 656.64,Z 339.431,A -85,B 0,C 180,E1 31306.438,E2 31306.438} C_VEL
LIN {X 0,Y 656.707,Z 339.425,A -85,B 0,C 180,E1 31303.549,E2 31303.549} C_VEL
LIN {X 0,Y 656.641,Z 339.421,A -85,B 0,C 180,E1 31300.52,E2 31300.52} C_VEL
LIN {X 0,Y 656.676,Z 339.434,A -85,B 0,C 180,E1 31297.719,E2 31297.719} C_VEL
LIN {X 0,Y 656.65,Z 339.43,A -85,B 0,C 180,E1 31294.57,E2 31294.57} C_VEL
LIN {X 0,Y 656.655,Z 339.429,A -85,B 0,C 180,E1 31291.833,E2 31291.833} C_VEL
LIN {X 0,Y 656.659,Z 339.43,A -85,B 0,C 180,E1 31288.617,E2 31288.617} C_VEL
LIN {X 0,Y 656.643,Z 339.434,A -85,B 0,C 180,E1 31285.919,E2 31285.919} C_VEL
LIN {X 0,Y 656.707,Z 339.429,A -85,B 0,C 180,E1 31282.919,E2 31282.919} C_VEL
LIN {X 0,Y 656.639,Z 339.434,A -85,B 0,C 180,E1 31280.014,E2 31280.014} C_VEL
LIN {X 0,Y 656.706,Z 339.421,A -85,B 0,C 180,E1 31277.085,E2 31277.085} C_VEL
LIN {X 0,Y 656.641,Z 339.434,A -85,B 0,C 180,E1 31274.05,E2 31274.05} C_VEL
LIN {X 0,Y 656.657,Z 339.564,A -85,B 0,C 180,E1 31271.831,E2 31271.831} C_VEL
LIN {X 0,Y 665.444,Z 362.462,A -85,B 0,C 180,E1 31269.3,E2 31269.3} C_VEL
LIN {X 0,Y 668.552,Z 371.163,A -85,B 0,C 180,E1 31268.399,E2 31268.399} C_VEL
LIN {X 0,Y 668.496,Z 376.599,A -85,B 0,C 180,E1 31268.008,E2 31268.008} C_VEL
LIN {X 0,Y 674.269,Z 401.065,A -85,B 0,C 180,E1 31267.308,E2 31267.308} C_VEL
LIN {X 0,Y 671.315,Z 665.727,A -85,B 0,C 180,E1 31264.087,E2 31264.087} C_VEL
LIN {X 0,Y 670.159,Z 767.71,A -85,B 0,C 180,E1 31262.844,E2 31262.844} C_VEL
LIN {X 0,Y 669.461,Z 793.012,A -85,B 0,C 180,E1 31262.384,E2 31262.384} C_VEL
LIN {X 0,Y 668.687,Z 814.008,A -85,B 0,C 180,E1 31261.869,E2 31261.869} C_VEL
LIN {X 0,Y 667.732,Z 837.259,A -85,B 0,C 180,E1 31261.156,E2 31261.156} C_VEL
LIN {X 0,Y 666.67,Z 858.208,A -85,B 0,C 180,E1 31260.361,E2 31260.361} C_VEL
LIN {X 0,Y 665.63,Z 878.27,A -85,B 0,C 180,E1 31259.47,E2 31259.47} C_VEL
LIN {X 0,Y 664.254,Z 901.417,A -85,B 0,C 180,E1 31258.261,E2 31258.261} C_VEL
LIN {X 0,Y 663.095,Z 920.728,A -85,B 0,C 180,E1 31257.09,E2 31257.09} C_VEL
LIN {X 0,Y 661.775,Z 942.003,A -85,B 0,C 180,E1 31255.602,E2 31255.602} C_VEL
LIN {X 0,Y 660.695,Z 959.4,A -85,B 0,C 180,E1 31254.213,E2 31254.213} C_VEL
LIN {X 0,Y 659.552,Z 978.604,A -85,B 0,C 180,E1 31252.46,E2 31252.46} C_VEL
LIN {X 0,Y 658.706,Z 993.631,A -85,B 0,C 180,E1 31250.899,E2 31250.899} C_VEL
LIN {X 0,Y 657.857,Z 1009.82,A -85,B 0,C 180,E1 31248.982,E2 31248.982} C_VEL
LIN {X 0,Y 657.284,Z 1022.521,A -85,B 0,C 180,E1 31247.256,E2 31247.256} C_VEL
LIN {X 0,Y 656.745,Z 1035.972,A -85,B 0,C 180,E1 31245.145,E2 31245.145} C_VEL
LIN {X 0,Y 656.42,Z 1046.022,A -85,B 0,C 180,E1 31243.298,E2 31243.298} C_VEL
LIN {X 0,Y 656.155,Z 1056.164,A -85,B 0,C 180,E1 31241.076,E2 31241.076} C_VEL
LIN {X 0,Y 656.032,Z 1063.12,A -85,B 0,C 180,E1 31239.209,E2 31239.209} C_VEL
LIN {X 0,Y 655.964,Z 1069.45,A -85,B 0,C 180,E1 31237.092,E2 31237.092} C_VEL
LIN {X 0,Y 655.926,Z 1073.816,A -85,B 0,C 180,E1 31235.072,E2 31235.072} C_VEL
LIN {X 0,Y 655.917,Z 1076.8,A -85,B 0,C 180,E1 31233.058,E2 31233.058} C_VEL
LIN {X 0,Y 655.906,Z 1078.283,A -85,B 0,C 180,E1 31230.873,E2 31230.873} C_VEL
LIN {X 0,Y 655.91,Z 1078.26,A -85,B 0,C 180,E1 31229.039,E2 31229.039} C_VEL
LIN {X 0,Y 655.917,Z 1076.574,A -85,B 0,C 180,E1 31226.767,E2 31226.767} C_VEL
LIN {X 0,Y 655.925,Z 1073.655,A -85,B 0,C 180,E1 31224.84,E2 31224.84} C_VEL
LIN {X 0,Y 655.96,Z 1069.016,A -85,B 0,C 180,E1 31222.732,E2 31222.732} C_VEL
LIN {X 0,Y 656.041,Z 1062.816,A -85,B 0,C 180,E1 31220.703,E2 31220.703} C_VEL
LIN {X 0,Y 656.163,Z 1055.832,A -85,B 0,C 180,E1 31218.841,E2 31218.841} C_VEL
LIN {X 0,Y 656.42,Z 1046.025,A -85,B 0,C 180,E1 31216.702,E2 31216.702} C_VEL
LIN {X 0,Y 656.745,Z 1035.974,A -85,B 0,C 180,E1 31214.855,E2 31214.855} C_VEL
LIN {X 0,Y 657.284,Z 1022.523,A -85,B 0,C 180,E1 31212.744,E2 31212.744} C_VEL
LIN {X 0,Y 657.857,Z 1009.82,A -85,B 0,C 180,E1 31211.019,E2 31211.019} C_VEL
LIN {X 0,Y 658.706,Z 993.631,A -85,B 0,C 180,E1 31209.101,E2 31209.101} C_VEL
LIN {X 0,Y 659.552,Z 978.605,A -85,B 0,C 180,E1 31207.54,E2 31207.54} C_VEL
LIN {X 0,Y 660.724,Z 958.846,A -85,B 0,C 180,E1 31205.741,E2 31205.741} C_VEL
LIN {X 0,Y 661.83,Z 941.235,A -85,B 0,C 180,E1 31204.34,E2 31204.34} C_VEL
LIN {X 0,Y 663.131,Z 919.985,A -85,B 0,C 180,E1 31202.863,E2 31202.863} C_VEL
LIN {X 0,Y 664.304,Z 900.683,A -85,B 0,C 180,E1 31201.697,E2 31201.697} C_VEL
LIN {X 0,Y 665.679,Z 877.27,A -85,B 0,C 180,E1 31200.483,E2 31200.483} C_VEL
LIN {X 0,Y 666.708,Z 857.462,A -85,B 0,C 180,E1 31199.608,E2 31199.608} C_VEL
LIN {X 0,Y 667.886,Z 833.797,A -85,B 0,C 180,E1 31198.729,E2 31198.729} C_VEL
LIN {X 0,Y 668.755,Z 812.386,A -85,B 0,C 180,E1 31198.087,E2 31198.087} C_VEL
LIN {X 0,Y 669.581,Z 790.077,A -85,B 0,C 180,E1 31197.551,E2 31197.551} C_VEL
LIN {X 0,Y 670.189,Z 765.252,A -85,B 0,C 180,E1 31197.121,E2 31197.121} C_VEL
LIN {X 0,Y 672.804,Z 526.404,A -85,B 0,C 180,E1 31194.226,E2 31194.226} C_VEL
LIN {X 0,Y 674.093,Z 399.551,A -85,B 0,C 180,E1 31192.661,E2 31192.661} C_VEL
LIN {X 0,Y 668.399,Z 375.76,A -85,B 0,C 180,E1 31191.951,E2 31191.951} C_VEL
LIN {X 0,Y 668.438,Z 370.567,A -85,B 0,C 180,E1 31191.544,E2 31191.544} C_VEL
LIN {X 0,Y 660.208,Z 348.828,A -85,B 0,C 180,E1 31189.223,E2 31189.223} C_VEL
LIN {X 0,Y 656.64,Z 339.439,A -85,B 0,C 180,E1 31188.167,E2 31188.167} C_VEL
LIN {X 0,Y 656.699,Z 339.433,A -85,B 0,C 180,E1 31185.296,E2 31185.296} C_VEL
LIN {X 0,Y 656.645,Z 339.436,A -85,B 0,C 180,E1 31182.265,E2 31182.265} C_VEL
LIN {X 0,Y 656.66,Z 339.425,A -85,B 0,C 180,E1 31179.53,E2 31179.53} C_VEL
LIN {X 0,Y 656.656,Z 339.435,A -85,B 0,C 180,E1 31176.323,E2 31176.323} C_VEL
LIN {X 0,Y 656.648,Z 339.427,A -85,B 0,C 180,E1 31173.599,E2 31173.599} C_VEL
LIN {X 0,Y 656.683,Z 339.427,A -85,B 0,C 180,E1 31170.467,E2 31170.467} C_VEL
LIN {X 0,Y 656.642,Z 339.423,A -85,B 0,C 180,E1 31167.674,E2 31167.674} C_VEL
LIN {X 0,Y 656.711,Z 339.428,A -85,B 0,C 180,E1 31164.636,E2 31164.636} C_VEL
LIN {X 0,Y 656.639,Z 339.431,A -85,B 0,C 180,E1 31161.717,E2 31161.717} C_VEL
LIN {X 0,Y 656.699,Z 339.419,A -85,B 0,C 180,E1 31158.832,E2 31158.832} C_VEL
LIN {X 0,Y 656.646,Z 339.428,A -85,B 0,C 180,E1 31155.77,E2 31155.77} C_VEL
LIN {X 0,Y 656.673,Z 339.424,A -85,B 0,C 180,E1 31152.966,E2 31152.966} C_VEL
LIN {X 0,Y 656.653,Z 339.421,A -85,B 0,C 180,E1 31149.819,E2 31149.819} C_VEL
LIN {X 0,Y 656.653,Z 339.429,A -85,B 0,C 180,E1 31147.085,E2 31147.085} C_VEL
LIN {X 0,Y 656.673,Z 339.425,A -85,B 0,C 180,E1 31143.929,E2 31143.929} C_VEL
LIN {X 0,Y 656.646,Z 339.429,A -85,B 0,C 180,E1 31141.134,E2 31141.134} C_VEL
LIN {X 0,Y 656.702,Z 339.423,A -85,B 0,C 180,E1 31138.08,E2 31138.08} C_VEL
LIN {X 0,Y 656.642,Z 339.426,A -85,B 0,C 180,E1 31135.196,E2 31135.196} C_VEL
LIN {X 0,Y 656.712,Z 339.424,A -85,B 0,C 180,E1 31132.212,E2 31132.212} C_VEL
LIN {X 0,Y 656.642,Z 339.419,A -85,B 0,C 180,E1 31129.205,E2 31129.205} C_VEL
LIN {X 0,Y 656.704,Z 339.427,A -85,B 0,C 180,E1 31126.267,E2 31126.267} C_VEL
LIN {X 0,Y 656.649,Z 339.428,A -85,B 0,C 180,E1 31123.274,E2 31123.274} C_VEL
LIN {X 0,Y 656.668,Z 339.428,A -85,B 0,C 180,E1 31120.481,E2 31120.481} C_VEL
LIN {X 0,Y 656.662,Z 339.433,A -85,B 0,C 180,E1 31117.331,E2 31117.331} C_VEL
LIN {X 0,Y 656.65,Z 339.419,A -85,B 0,C 180,E1 31114.57,E2 31114.57} C_VEL
LIN {X 0,Y 656.683,Z 339.425,A -85,B 0,C 180,E1 31111.438,E2 31111.438} C_VEL
LIN {X 0,Y 656.647,Z 339.431,A -85,B 0,C 180,E1 31108.616,E2 31108.616} C_VEL
LIN {X 0,Y 656.708,Z 339.425,A -85,B 0,C 180,E1 31105.606,E2 31105.606} C_VEL
LIN {X 0,Y 656.645,Z 339.43,A -85,B 0,C 180,E1 31102.642,E2 31102.642} C_VEL
LIN {X 0,Y 656.644,Z 339.428,A -85,B 0,C 180,E1 31100.617,E2 31100.617} C_VEL
LIN {X 0,Y 655.666,Z 339.552,A -85,B 0,C 180,E1 31099.946,E2 31099.946} C_VEL
LIN {X 0,Y 649.315,Z 340.354,A -85,B 0,C 180,E1 31098.061,E2 31098.061} C_VEL
LIN {X 0,Y 648.773,Z 340.412,A -85,B 0,C 180,E1 31097.571,E2 31097.571} C_VEL
LIN {X 0,Y 648.706,Z 340.41,A -85,B 0,C 180,E1 31094.593,E2 31094.593} C_VEL
LIN {X 0,Y 648.771,Z 340.413,A -85,B 0,C 180,E1 31091.626,E2 31091.626} C_VEL
LIN {X 0,Y 648.711,Z 340.428,A -85,B 0,C 180,E1 31088.605,E2 31088.605} C_VEL
LIN {X 0,Y 648.725,Z 340.49,A -85,B 0,C 180,E1 31088.119,E2 31088.119} C_VEL
LIN {X 0,Y 652.031,Z 349.362,A -85,B 0,C 180,E1 31087.097,E2 31087.097} C_VEL
LIN {X 0,Y 664.392,Z 369.862,A -85,B 0,C 180,E1 31085.954,E2 31085.954} C_VEL
LIN {X 0,Y 667.91,Z 376.435,A -85,B 0,C 180,E1 31085.629,E2 31085.629} C_VEL
LIN {X 0,Y 664.987,Z 613.857,A -85,B 0,C 180,E1 31082.7,E2 31082.7} C_VEL
LIN {X 0,Y 663.442,Z 737.836,A -85,B 0,C 180,E1 31081.175,E2 31081.175} C_VEL
LIN {X 0,Y 662.693,Z 763.181,A -85,B 0,C 180,E1 31080.709,E2 31080.709} C_VEL
LIN {X 0,Y 661.868,Z 783.905,A -85,B 0,C 180,E1 31080.197,E2 31080.197} C_VEL
LIN {X 0,Y 660.864,Z 806.43,A -85,B 0,C 180,E1 31079.504,E2 31079.504} C_VEL
LIN {X 0,Y 659.611,Z 829.135,A -85,B 0,C 180,E1 31078.634,E2 31078.634} C_VEL
LIN {X 0,Y 658.444,Z 850.054,A -85,B 0,C 180,E1 31077.69,E2 31077.69} C_VEL
LIN {X 0,Y 656.995,Z 872.245,A -85,B 0,C 180,E1 31076.506,E2 31076.506} C_VEL
LIN {X 0,Y 655.751,Z 891.2,A -85,B 0,C 180,E1 31075.341,E2 31075.341} C_VEL
LIN {X 0,Y 654.372,Z 911.773,A -85,B 0,C 180,E1 31073.886,E2 31073.886} C_VEL
LIN {X 0,Y 653.2,Z 928.979,A -85,B 0,C 180,E1 31072.5,E2 31072.5} C_VEL
LIN {X 0,Y 651.965,Z 948.038,A -85,B 0,C 180,E1 31070.749,E2 31070.749} C_VEL
LIN {X 0,Y 651.012,Z 963.172,A -85,B 0,C 180,E1 31069.164,E2 31069.164} C_VEL
LIN {X 0,Y 650.073,Z 979.79,A -85,B 0,C 180,E1 31067.177,E2 31067.177} C_VEL
LIN {X 0,Y 649.433,Z 992.376,A -85,B 0,C 180,E1 31065.448,E2 31065.448} C_VEL
LIN {X 0,Y 648.851,Z 1005.546,A -85,B 0,C 180,E1 31063.365,E2 31063.365} C_VEL
LIN {X 0,Y 648.499,Z 1015.294,A -85,B 0,C 180,E1 31061.563,E2 31061.563} C_VEL
LIN {X 0,Y 648.228,Z 1024.856,A -85,B 0,C 180,E1 31059.5,E2 31059.5} C_VEL
LIN {X 0,Y 648.057,Z 1032.549,A -85,B 0,C 180,E1 31057.447,E2 31057.447} C_VEL
LIN {X 0,Y 647.956,Z 1038.766,A -85,B 0,C 180,E1 31055.401,E2 31055.401} C_VEL
LIN {X 0,Y 647.917,Z 1043.485,A -85,B 0,C 180,E1 31053.273,E2 31053.273} C_VEL
LIN {X 0,Y 647.912,Z 1046.338,A -85,B 0,C 180,E1 31051.415,E2 31051.415} C_VEL
LIN {X 0,Y 647.909,Z 1048.189,A -85,B 0,C 180,E1 31049.204,E2 31049.204} C_VEL
LIN {X 0,Y 647.897,Z 1048.331,A -85,B 0,C 180,E1 31047.258,E2 31047.258} C_VEL
LIN {X 0,Y 647.897,Z 1047.231,A -85,B 0,C 180,E1 31045.308,E2 31045.308} C_VEL
LIN {X 0,Y 647.916,Z 1044.293,A -85,B 0,C 180,E1 31043.086,E2 31043.086} C_VEL
LIN {X 0,Y 647.938,Z 1040.673,A -85,B 0,C 180,E1 31041.302,E2 31041.302} C_VEL
LIN {X 0,Y 647.999,Z 1035.15,A -85,B 0,C 180,E1 31039.239,E2 31039.239} C_VEL
LIN {X 0,Y 648.144,Z 1027.81,A -85,B 0,C 180,E1 31037.159,E2 31037.159} C_VEL
LIN {X 0,Y 648.366,Z 1019.725,A -85,B 0,C 180,E1 31035.259,E2 31035.259} C_VEL
LIN {X 0,Y 648.748,Z 1008.485,A -85,B 0,C 180,E1 31033.064,E2 31033.064} C_VEL
LIN {X 0,Y 649.199,Z 997.43,A -85,B 0,C 180,E1 31031.222,E2 31031.222} C_VEL
LIN {X 0,Y 649.881,Z 983.201,A -85,B 0,C 180,E1 31029.181,E2 31029.181} C_VEL
LIN {X 0,Y 650.668,Z 969.379,A -85,B 0,C 180,E1 31027.454,E2 31027.454} C_VEL
LIN {X 0,Y 651.687,Z 952.296,A -85,B 0,C 180,E1 31025.589,E2 31025.589} C_VEL
LIN {X 0,Y 652.723,Z 936.319,A -85,B 0,C 180,E1 31024.055,E2 31024.055} C_VEL
LIN {X 0,Y 654.057,Z 916.102,A -85,B 0,C 180,E1 31022.356,E2 31022.356} C_VEL
LIN {X 0,Y 655.311,Z 897.949,A -85,B 0,C 180,E1 31021.024,E2 31021.024} C_VEL
LIN {X 0,Y 656.737,Z 876.257,A -85,B 0,C 180,E1 31019.637,E2 31019.637} C_VEL
LIN {X 0,Y 657.95,Z 857.206,A -85,B 0,C 180,E1 31018.583,E2 31018.583} C_VEL
LIN {X 0,Y 659.382,Z 833.782,A -85,B 0,C 180,E1 31017.472,E2 31017.472} C_VEL
LIN {X 0,Y 660.484,Z 813.484,A -85,B 0,C 180,E1 31016.665,E2 31016.665} C_VEL
LIN {X 0,Y 661.599,Z 790.536,A -85,B 0,C 180,E1 31015.896,E2 31015.896} C_VEL
LIN {X 0,Y 662.533,Z 766.989,A -85,B 0,C 180,E1 31015.286,E2 31015.286} C_VEL
LIN {X 0,Y 663.294,Z 744.574,A -85,B 0,C 180,E1 31014.841,E2 31014.841} C_VEL
LIN {X 0,Y 663.855,Z 710.877,A -85,B 0,C 180,E1 31014.387,E2 31014.387} C_VEL
LIN {X 0,Y 666.921,Z 456.239,A -85,B 0,C 180,E1 31011.274,E2 31011.274} C_VEL
LIN {X 0,Y 667.73,Z 375.714,A -85,B 0,C 180,E1 31010.259,E2 31010.259} C_VEL
LIN {X 0,Y 657.19,Z 357.792,A -85,B 0,C 180,E1 31009.295,E2 31009.295} C_VEL
LIN {X 0,Y 651.704,Z 348.634,A -85,B 0,C 180,E1 31008.746,E2 31008.746} C_VEL
LIN {X 0,Y 648.713,Z 340.425,A -85,B 0,C 180,E1 31007.747,E2 31007.747} C_VEL
LIN {X 0,Y 648.736,Z 340.421,A -85,B 0,C 180,E1 31004.903,E2 31004.903} C_VEL
LIN {X 0,Y 648.717,Z 340.413,A -85,B 0,C 180,E1 31001.748,E2 31001.748} C_VEL
LIN {X 0,Y 648.719,Z 340.416,A -85,B 0,C 180,E1 30998.967,E2 30998.967} C_VEL
LIN {X 0,Y 648.722,Z 340.393,A -85,B 0,C 180,E1 30995.744,E2 30995.744} C_VEL
LIN {X 0,Y 648.713,Z 340.422,A -85,B 0,C 180,E1 30992.963,E2 30992.963} C_VEL
LIN {X 0,Y 648.744,Z 340.417,A -85,B 0,C 180,E1 30989.804,E2 30989.804} C_VEL
LIN {X 0,Y 648.707,Z 340.421,A -85,B 0,C 180,E1 30987.013,E2 30987.013} C_VEL
LIN {X 0,Y 648.768,Z 340.418,A -85,B 0,C 180,E1 30983.945,E2 30983.945} C_VEL
LIN {X 0,Y 648.704,Z 340.414,A -85,B 0,C 180,E1 30981.047,E2 30981.047} C_VEL
LIN {X 0,Y 648.767,Z 340.412,A -85,B 0,C 180,E1 30978.139,E2 30978.139} C_VEL
LIN {X 0,Y 648.705,Z 340.418,A -85,B 0,C 180,E1 30975.099,E2 30975.099} C_VEL
LIN {X 0,Y 648.743,Z 340.42,A -85,B 0,C 180,E1 30972.267,E2 30972.267} C_VEL
LIN {X 0,Y 648.711,Z 340.415,A -85,B 0,C 180,E1 30969.135,E2 30969.135} C_VEL
LIN {X 0,Y 648.722,Z 340.421,A -85,B 0,C 180,E1 30966.372,E2 30966.372} C_VEL
LIN {X 0,Y 648.722,Z 340.418,A -85,B 0,C 180,E1 30963.181,E2 30963.181} C_VEL
LIN {X 0,Y 648.709,Z 340.415,A -85,B 0,C 180,E1 30960.442,E2 30960.442} C_VEL
LIN {X 0,Y 648.751,Z 340.408,A -85,B 0,C 180,E1 30957.35,E2 30957.35} C_VEL
LIN {X 0,Y 648.703,Z 340.421,A -85,B 0,C 180,E1 30954.516,E2 30954.516} C_VEL
LIN {X 0,Y 648.776,Z 340.417,A -85,B 0,C 180,E1 30951.581,E2 30951.581} C_VEL
LIN {X 0,Y 648.703,Z 340.409,A -85,B 0,C 180,E1 30948.611,E2 30948.611} C_VEL
LIN {X 0,Y 648.757,Z 340.418,A -85,B 0,C 180,E1 30945.724,E2 30945.724} C_VEL
LIN {X 0,Y 648.712,Z 340.418,A -85,B 0,C 180,E1 30942.694,E2 30942.694} C_VEL
LIN {X 0,Y 648.722,Z 340.412,A -85,B 0,C 180,E1 30939.896,E2 30939.896} C_VEL
LIN {X 0,Y 648.715,Z 340.41,A -85,B 0,C 180,E1 30936.664,E2 30936.664} C_VEL
LIN {X 0,Y 648.712,Z 340.422,A -85,B 0,C 180,E1 30933.942,E2 30933.942} C_VEL
LIN {X 0,Y 648.733,Z 340.417,A -85,B 0,C 180,E1 30930.752,E2 30930.752} C_VEL
LIN {X 0,Y 648.705,Z 340.422,A -85,B 0,C 180,E1 30927.968,E2 30927.968} C_VEL
LIN {X 0,Y 648.762,Z 340.42,A -85,B 0,C 180,E1 30924.909,E2 30924.909} C_VEL
LIN {X 0,Y 648.7,Z 340.421,A -85,B 0,C 180,E1 30922.047,E2 30922.047} C_VEL
LIN {X 0,Y 648.775,Z 340.418,A -85,B 0,C 180,E1 30919.079,E2 30919.079} C_VEL
LIN {X 0,Y 648.702,Z 340.422,A -85,B 0,C 180,E1 30916.04,E2 30916.04} C_VEL
LIN {X 0,Y 648.75,Z 340.417,A -85,B 0,C 180,E1 30913.182,E2 30913.182} C_VEL
LIN {X 0,Y 648.729,Z 340.449,A -85,B 0,C 180,E1 30912.373,E2 30912.373} C_VEL
LIN {X 0,Y 651.433,Z 347.434,A -85,B 0,C 180,E1 30911.559,E2 30911.559} C_VEL
LIN {X 0,Y 659.934,Z 369.917,A -85,B 0,C 180,E1 30909.072,E2 30909.072} C_VEL
LIN {X 0,Y 661.535,Z 374.738,A -85,B 0,C 180,E1 30908.576,E2 30908.576} C_VEL
LIN {X 0,Y 661.641,Z 376.516,A -85,B 0,C 180,E1 30908.472,E2 30908.472} C_VEL
LIN {X 0,Y 667.865,Z 402.872,A -85,B 0,C 180,E1 30907.701,E2 30907.701} C_VEL
LIN {X 0,Y 664.643,Z 668.434,A -85,B 0,C 180,E1 30904.44,E2 30904.44} C_VEL
LIN {X 0,Y 663.414,Z 767.858,A -85,B 0,C 180,E1 30903.215,E2 30903.215} C_VEL
LIN {X 0,Y 662.658,Z 793.274,A -85,B 0,C 180,E1 30902.748,E2 30902.748} C_VEL
LIN {X 0,Y 661.842,Z 814.057,A -85,B 0,C 180,E1 30902.235,E2 30902.235} C_VEL
LIN {X 0,Y 660.815,Z 837.255,A -85,B 0,C 180,E1 30901.519,E2 30901.519} C_VEL
LIN {X 0,Y 659.604,Z 859.334,A -85,B 0,C 180,E1 30900.67,E2 30900.67} C_VEL
LIN {X 0,Y 658.379,Z 881.272,A -85,B 0,C 180,E1 30899.676,E2 30899.676} C_VEL
LIN {X 0,Y 656.935,Z 903.117,A -85,B 0,C 180,E1 30898.5,E2 30898.5} C_VEL
LIN {X 0,Y 655.617,Z 923.649,A -85,B 0,C 180,E1 30897.228,E2 30897.228} C_VEL
LIN {X 0,Y 654.268,Z 943.217,A -85,B 0,C 180,E1 30895.821,E2 30895.821} C_VEL
LIN {X 0,Y 653.066,Z 961.203,A -85,B 0,C 180,E1 30894.357,E2 30894.357} C_VEL
LIN {X 0,Y 651.925,Z 978.603,A -85,B 0,C 180,E1 30892.737,E2 30892.737} C_VEL
LIN {X 0,Y 650.992,Z 993.629,A -85,B 0,C 180,E1 30891.158,E2 30891.158} C_VEL
LIN {X 0,Y 650.06,Z 1010.027,A -85,B 0,C 180,E1 30889.191,E2 30889.191} C_VEL
LIN {X 0,Y 649.428,Z 1022.519,A -85,B 0,C 180,E1 30887.472,E2 30887.472} C_VEL
LIN {X 0,Y 648.846,Z 1035.767,A -85,B 0,C 180,E1 30885.37,E2 30885.37} C_VEL
LIN {X 0,Y 648.494,Z 1045.563,A -85,B 0,C 180,E1 30883.554,E2 30883.554} C_VEL
LIN {X 0,Y 648.208,Z 1055.479,A -85,B 0,C 180,E1 30881.388,E2 30881.388} C_VEL
LIN {X 0,Y 648.055,Z 1062.514,A -85,B 0,C 180,E1 30879.503,E2 30879.503} C_VEL
LIN {X 0,Y 647.954,Z 1068.761,A -85,B 0,C 180,E1 30877.448,E2 30877.448} C_VEL
LIN {X 0,Y 647.924,Z 1073.496,A -85,B 0,C 180,E1 30875.313,E2 30875.313} C_VEL
LIN {X 0,Y 647.913,Z 1076.35,A -85,B 0,C 180,E1 30873.451,E2 30873.451} C_VEL
LIN {X 0,Y 647.905,Z 1078.192,A -85,B 0,C 180,E1 30871.238,E2 30871.238} C_VEL
LIN {X 0,Y 647.897,Z 1078.328,A -85,B 0,C 180,E1 30869.293,E2 30869.293} C_VEL
LIN {X 0,Y 647.907,Z 1077.157,A -85,B 0,C 180,E1 30867.258,E2 30867.258} C_VEL
LIN {X 0,Y 647.925,Z 1074.133,A -85,B 0,C 180,E1 30865.042,E2 30865.042} C_VEL
LIN {X 0,Y 647.94,Z 1070.276,A -85,B 0,C 180,E1 30863.176,E2 30863.176} C_VEL
LIN {X 0,Y 648.021,Z 1064.006,A -85,B 0,C 180,E1 30860.938,E2 30860.938} C_VEL
LIN {X 0,Y 648.158,Z 1057.25,A -85,B 0,C 180,E1 30859.062,E2 30859.062} C_VEL
LIN {X 0,Y 648.402,Z 1048.623,A -85,B 0,C 180,E1 30857.059,E2 30857.059} C_VEL
LIN {X 0,Y 648.764,Z 1037.835,A -85,B 0,C 180,E1 30854.994,E2 30854.994} C_VEL
LIN {X 0,Y 649.259,Z 1026.235,A -85,B 0,C 180,E1 30853.078,E2 30853.078} C_VEL
LIN {X 0,Y 649.923,Z 1012.35,A -85,B 0,C 180,E1 30851.114,E2 30851.114} C_VEL
LIN {X 0,Y 650.773,Z 997.755,A -85,B 0,C 180,E1 30849.305,E2 30849.305} C_VEL
LIN {X 0,Y 651.742,Z 981.381,A -85,B 0,C 180,E1 30847.542,E2 30847.542} C_VEL
LIN {X 0,Y 652.839,Z 964.771,A -85,B 0,C 180,E1 30845.958,E2 30845.958} C_VEL
LIN {X 0,Y 654.088,Z 945.648,A -85,B 0,C 180,E1 30844.366,E2 30844.366} C_VEL
LIN {X 0,Y 655.324,Z 927.727,A -85,B 0,C 180,E1 30843.053,E2 30843.053} C_VEL
LIN {X 0,Y 656.777,Z 905.546,A -85,B 0,C 180,E1 30841.641,E2 30841.641} C_VEL
LIN {X 0,Y 658.052,Z 885.844,A -85,B 0,C 180,E1 30840.558,E2 30840.558} C_VEL
LIN {X 0,Y 659.456,Z 862.306,A -85,B 0,C 180,E1 30839.455,E2 30839.455} C_VEL
LIN {X 0,Y 660.538,Z 842.394,A -85,B 0,C 180,E1 30838.67,E2 30838.67} C_VEL
LIN {X 0,Y 661.643,Z 818.851,A -85,B 0,C 180,E1 30837.895,E2 30837.895} C_VEL
LIN {X 0,Y 662.54,Z 796.094,A -85,B 0,C 180,E1 30837.315,E2 30837.315} C_VEL
LIN {X 0,Y 663.333,Z 772.593,A -85,B 0,C 180,E1 30836.856,E2 30836.856} C_VEL
LIN {X 0,Y 663.909,Z 733.531,A -85,B 0,C 180,E1 30836.348,E2 30836.348} C_VEL
LIN {X 0,Y 666.864,Z 481.94,A -85,B 0,C 180,E1 30833.278,E2 30833.278} C_VEL
LIN {X 0,Y 667.697,Z 401.371,A -85,B 0,C 180,E1 30832.268,E2 30832.268} C_VEL
LIN {X 0,Y 661.514,Z 375.529,A -85,B 0,C 180,E1 30831.483,E2 30831.483} C_VEL
LIN {X 0,Y 661.214,Z 373.349,A -85,B 0,C 180,E1 30831.288,E2 30831.288} C_VEL
LIN {X 0,Y 653.386,Z 352.647,A -85,B 0,C 180,E1 30829.051,E2 30829.051} C_VEL
LIN {X 0,Y 648.724,Z 340.426,A -85,B 0,C 180,E1 30827.658,E2 30827.658} C_VEL
LIN {X 0,Y 648.719,Z 340.427,A -85,B 0,C 180,E1 30824.469,E2 30824.469} C_VEL
LIN {X 0,Y 648.708,Z 340.423,A -85,B 0,C 180,E1 30821.749,E2 30821.749} C_VEL
LIN {X 0,Y 648.761,Z 340.422,A -85,B 0,C 180,E1 30818.737,E2 30818.737} C_VEL
LIN {X 0,Y 648.702,Z 340.422,A -85,B 0,C 180,E1 30815.83,E2 30815.83} C_VEL
LIN {X 0,Y 648.772,Z 340.416,A -85,B 0,C 180,E1 30812.854,E2 30812.854} C_VEL
LIN {X 0,Y 648.703,Z 340.419,A -85,B 0,C 180,E1 30809.859,E2 30809.859} C_VEL
LIN {X 0,Y 648.756,Z 340.407,A -85,B 0,C 180,E1 30807.021,E2 30807.021} C_VEL
LIN {X 0,Y 648.706,Z 340.412,A -85,B 0,C 180,E1 30803.932,E2 30803.932} C_VEL
LIN {X 0,Y 648.727,Z 340.418,A -85,B 0,C 180,E1 30801.173,E2 30801.173} C_VEL
LIN {X 0,Y 648.715,Z 340.421,A -85,B 0,C 180,E1 30797.955,E2 30797.955} C_VEL
LIN {X 0,Y 648.717,Z 340.415,A -85,B 0,C 180,E1 30795.19,E2 30795.19} C_VEL
LIN {X 0,Y 648.729,Z 340.422,A -85,B 0,C 180,E1 30792.01,E2 30792.01} C_VEL
LIN {X 0,Y 648.707,Z 340.407,A -85,B 0,C 180,E1 30789.224,E2 30789.224} C_VEL
LIN {X 0,Y 648.763,Z 340.418,A -85,B 0,C 180,E1 30786.193,E2 30786.193} C_VEL
LIN {X 0,Y 648.703,Z 340.416,A -85,B 0,C 180,E1 30783.269,E2 30783.269} C_VEL
LIN {X 0,Y 648.775,Z 340.412,A -85,B 0,C 180,E1 30780.265,E2 30780.265} C_VEL
LIN {X 0,Y 648.704,Z 340.42,A -85,B 0,C 180,E1 30777.261,E2 30777.261} C_VEL
LIN {X 0,Y 648.768,Z 340.409,A -85,B 0,C 180,E1 30774.339,E2 30774.339} C_VEL
LIN {X 0,Y 648.706,Z 340.421,A -85,B 0,C 180,E1 30771.312,E2 30771.312} C_VEL
LIN {X 0,Y 648.747,Z 340.403,A -85,B 0,C 180,E1 30768.442,E2 30768.442} C_VEL
LIN {X 0,Y 648.713,Z 340.417,A -85,B 0,C 180,E1 30765.358,E2 30765.358} C_VEL
LIN {X 0,Y 648.725,Z 340.413,A -85,B 0,C 180,E1 30762.568,E2 30762.568} C_VEL
LIN {X 0,Y 648.718,Z 340.411,A -85,B 0,C 180,E1 30759.323,E2 30759.323} C_VEL
LIN {X 0,Y 648.717,Z 340.419,A -85,B 0,C 180,E1 30756.568,E2 30756.568} C_VEL
LIN {X 0,Y 648.732,Z 340.423,A -85,B 0,C 180,E1 30753.351,E2 30753.351} C_VEL
LIN {X 0,Y 648.712,Z 340.409,A -85,B 0,C 180,E1 30750.548,E2 30750.548} C_VEL
LIN {X 0,Y 648.756,Z 340.414,A -85,B 0,C 180,E1 30747.459,E2 30747.459} C_VEL
LIN {X 0,Y 648.71,Z 340.42,A -85,B 0,C 180,E1 30744.581,E2 30744.581} C_VEL
LIN {X 0,Y 648.773,Z 340.422,A -85,B 0,C 180,E1 30741.49,E2 30741.49} C_VEL
LIN {X 0,Y 648.707,Z 340.424,A -85,B 0,C 180,E1 30738.605,E2 30738.605} C_VEL
LIN {X 0,Y 648.773,Z 340.412,A -85,B 0,C 180,E1 30737.571,E2 30737.571} C_VEL
LIN {X 0,Y 647.756,Z 340.524,A -85,B 0,C 180,E1 30736.891,E2 30736.891} C_VEL
LIN {X 0,Y 641.295,Z 341.322,A -85,B 0,C 180,E1 30734.984,E2 30734.984} C_VEL
LIN {X 0,Y 640.768,Z 341.399,A -85,B 0,C 180,E1 30734.487,E2 30734.487} C_VEL
LIN {X 0,Y 640.837,Z 341.402,A -85,B 0,C 180,E1 30731.501,E2 30731.501} C_VEL
LIN {X 0,Y 640.79,Z 341.545,A -85,B 0,C 180,E1 30728.635,E2 30728.635} C_VEL
LIN {X 0,Y 643.877,Z 349.627,A -85,B 0,C 180,E1 30727.682,E2 30727.682} C_VEL
LIN {X 0,Y 658.867,Z 374.361,A -85,B 0,C 180,E1 30726.271,E2 30726.271} C_VEL
LIN {X 0,Y 661.548,Z 379.54,A -85,B 0,C 180,E1 30726.017,E2 30726.017} C_VEL
LIN {X 0,Y 658.385,Z 617.08,A -85,B 0,C 180,E1 30723.06,E2 30723.06} C_VEL
LIN {X 0,Y 656.757,Z 738.068,A -85,B 0,C 180,E1 30721.557,E2 30721.557} C_VEL
LIN {X 0,Y 655.957,Z 763.521,A -85,B 0,C 180,E1 30721.085,E2 30721.085} C_VEL
LIN {X 0,Y 655.089,Z 784.002,A -85,B 0,C 180,E1 30720.575,E2 30720.575} C_VEL
LIN {X 0,Y 654.039,Z 806.034,A -85,B 0,C 180,E1 30719.893,E2 30719.893} C_VEL
LIN {X 0,Y 652.714,Z 827.923,A -85,B 0,C 180,E1 30719.052,E2 30719.052} C_VEL
LIN {X 0,Y 651.447,Z 848.647,A -85,B 0,C 180,E1 30718.113,E2 30718.113} C_VEL
LIN {X 0,Y 649.878,Z 871.49,A -85,B 0,C 180,E1 30716.894,E2 30716.894} C_VEL
LIN {X 0,Y 648.51,Z 890.461,A -85,B 0,C 180,E1 30715.723,E2 30715.723} C_VEL
LIN {X 0,Y 647.011,Z 911.25,A -85,B 0,C 180,E1 30714.246,E2 30714.246} C_VEL
LIN {X 0,Y 645.766,Z 928.204,A -85,B 0,C 180,E1 30712.87,E2 30712.87} C_VEL
LIN {X 0,Y 644.461,Z 946.619,A -85,B 0,C 180,E1 30711.177,E2 30711.177} C_VEL
LIN {X 0,Y 643.38,Z 962.356,A -85,B 0,C 180,E1 30709.52,E2 30709.52} C_VEL
LIN {X 0,Y 642.423,Z 977.898,A -85,B 0,C 180,E1 30707.668,E2 30707.668} C_VEL
LIN {X 0,Y 641.632,Z 991.301,A -85,B 0,C 180,E1 30705.826,E2 30705.826} C_VEL
LIN {X 0,Y 641.024,Z 1004.152,A -85,B 0,C 180,E1 30703.807,E2 30703.807} C_VEL
LIN {X 0,Y 640.573,Z 1014.97,A -85,B 0,C 180,E1 30701.799,E2 30701.799} C_VEL
LIN {X 0,Y 640.272,Z 1024.604,A -85,B 0,C 180,E1 30699.71,E2 30699.71} C_VEL
LIN {X 0,Y 640.067,Z 1032.335,A -85,B 0,C 180,E1 30697.63,E2 30697.63} C_VEL
LIN {X 0,Y 639.965,Z 1038.079,A -85,B 0,C 180,E1 30695.739,E2 30695.739} C_VEL
LIN {X 0,Y 639.916,Z 1043.212,A -85,B 0,C 180,E1 30693.494,E2 30693.494} C_VEL
LIN {X 0,Y 639.913,Z 1046.145,A -85,B 0,C 180,E1 30691.612,E2 30691.612} C_VEL
LIN {X 0,Y 639.9,Z 1048.112,A -85,B 0,C 180,E1 30689.463,E2 30689.463} C_VEL
LIN {X 0,Y 639.895,Z 1048.347,A -85,B 0,C 180,E1 30687.313,E2 30687.313} C_VEL
LIN {X 0,Y 639.898,Z 1047.279,A -85,B 0,C 180,E1 30685.339,E2 30685.339} C_VEL
LIN {X 0,Y 639.917,Z 1044.407,A -85,B 0,C 180,E1 30683.09,E2 30683.09} C_VEL
LIN {X 0,Y 639.946,Z 1040.613,A -85,B 0,C 180,E1 30681.192,E2 30681.192} C_VEL
LIN {X 0,Y 640.019,Z 1034.786,A -85,B 0,C 180,E1 30679.012,E2 30679.012} C_VEL
LIN {X 0,Y 640.168,Z 1027.729,A -85,B 0,C 180,E1 30677.002,E2 30677.002} C_VEL
LIN {X 0,Y 640.412,Z 1019.823,A -85,B 0,C 180,E1 30675.12,E2 30675.12} C_VEL
LIN {X 0,Y 640.82,Z 1008.851,A -85,B 0,C 180,E1 30672.942,E2 30672.942} C_VEL
LIN {X 0,Y 641.314,Z 997.845,A -85,B 0,C 180,E1 30671.077,E2 30671.077} C_VEL
LIN {X 0,Y 642.053,Z 983.699,A -85,B 0,C 180,E1 30669.011,E2 30669.011} C_VEL
LIN {X 0,Y 642.904,Z 969.922,A -85,B 0,C 180,E1 30667.262,E2 30667.262} C_VEL
LIN {X 0,Y 644.05,Z 952.357,A -85,B 0,C 180,E1 30665.315,E2 30665.315} C_VEL
LIN {X 0,Y 645.16,Z 936.633,A -85,B 0,C 180,E1 30663.787,E2 30663.787} C_VEL
LIN {X 0,Y 646.621,Z 916.353,A -85,B 0,C 180,E1 30662.061,E2 30662.061} C_VEL
LIN {X 0,Y 647.915,Z 898.903,A -85,B 0,C 180,E1 30660.762,E2 30660.762} C_VEL
LIN {X 0,Y 649.455,Z 877.42,A -85,B 0,C 180,E1 30659.363,E2 30659.363} C_VEL
LIN {X 0,Y 650.753,Z 858.498,A -85,B 0,C 180,E1 30658.299,E2 30658.299} C_VEL
LIN {X 0,Y 652.23,Z 836.818,A -85,B 0,C 180,E1 30657.237,E2 30657.237} C_VEL
LIN {X 0,Y 653.53,Z 814.727,A -85,B 0,C 180,E1 30656.337,E2 30656.337} C_VEL
LIN {X 0,Y 654.64,Z 793.649,A -85,B 0,C 180,E1 30655.615,E2 30655.615} C_VEL
LIN {X 0,Y 655.721,Z 768.897,A -85,B 0,C 180,E1 30654.946,E2 30654.946} C_VEL
LIN {X 0,Y 656.498,Z 747.393,A -85,B 0,C 180,E1 30654.506,E2 30654.506} C_VEL
LIN {X 0,Y 657.137,Z 716.349,A -85,B 0,C 180,E1 30654.066,E2 30654.066} C_VEL
LIN {X 0,Y 660.441,Z 462.018,A -85,B 0,C 180,E1 30650.929,E2 30650.929} C_VEL
LIN {X 0,Y 661.384,Z 378.795,A -85,B 0,C 180,E1 30649.872,E2 30649.872} C_VEL
LIN {X 0,Y 649.906,Z 359.323,A -85,B 0,C 180,E1 30648.793,E2 30648.793} C_VEL
LIN {X 0,Y 643.631,Z 348.945,A -85,B 0,C 180,E1 30648.152,E2 30648.152} C_VEL
LIN {X 0,Y 640.777,Z 341.41,A -85,B 0,C 180,E1 30647.19,E2 30647.19} C_VEL
LIN {X 0,Y 640.799,Z 341.403,A -85,B 0,C 180,E1 30644,E2 30644} C_VEL
LIN {X 0,Y 640.766,Z 341.392,A -85,B 0,C 180,E1 30641.187,E2 30641.187} C_VEL
LIN {X 0,Y 640.826,Z 341.406,A -85,B 0,C 180,E1 30638.15,E2 30638.15} C_VEL
LIN {X 0,Y 640.765,Z 341.385,A -85,B 0,C 180,E1 30635.157,E2 30635.157} C_VEL
LIN {X 0,Y 640.829,Z 341.399,A -85,B 0,C 180,E1 30632.087,E2 30632.087} C_VEL
LIN {X 0,Y 640.766,Z 341.409,A -85,B 0,C 180,E1 30629.135,E2 30629.135} C_VEL
LIN {X 0,Y 640.833,Z 341.403,A -85,B 0,C 180,E1 30626.204,E2 30626.204} C_VEL
LIN {X 0,Y 640.766,Z 341.41,A -85,B 0,C 180,E1 30623.156,E2 30623.156} C_VEL
LIN {X 0,Y 640.822,Z 341.407,A -85,B 0,C 180,E1 30620.267,E2 30620.267} C_VEL
LIN {X 0,Y 640.767,Z 341.404,A -85,B 0,C 180,E1 30617.153,E2 30617.153} C_VEL
LIN {X 0,Y 640.808,Z 341.403,A -85,B 0,C 180,E1 30614.273,E2 30614.273} C_VEL
LIN {X 0,Y 640.773,Z 341.406,A -85,B 0,C 180,E1 30611.157,E2 30611.157} C_VEL
LIN {X 0,Y 640.787,Z 341.408,A -85,B 0,C 180,E1 30608.344,E2 30608.344} C_VEL
LIN {X 0,Y 640.781,Z 341.402,A -85,B 0,C 180,E1 30605.193,E2 30605.193} C_VEL
LIN {X 0,Y 640.774,Z 341.41,A -85,B 0,C 180,E1 30602.415,E2 30602.415} C_VEL
LIN {X 0,Y 640.791,Z 341.407,A -85,B 0,C 180,E1 30599.195,E2 30599.195} C_VEL
LIN {X 0,Y 640.767,Z 341.402,A -85,B 0,C 180,E1 30596.421,E2 30596.421} C_VEL
LIN {X 0,Y 640.825,Z 341.394,A -85,B 0,C 180,E1 30593.37,E2 30593.37} C_VEL
LIN {X 0,Y 640.764,Z 341.41,A -85,B 0,C 180,E1 30590.475,E2 30590.475} C_VEL
LIN {X 0,Y 640.834,Z 341.405,A -85,B 0,C 180,E1 30587.474,E2 30587.474} C_VEL
LIN {X 0,Y 640.764,Z 341.398,A -85,B 0,C 180,E1 30584.524,E2 30584.524} C_VEL
LIN {X 0,Y 640.816,Z 341.405,A -85,B 0,C 180,E1 30581.628,E2 30581.628} C_VEL
LIN {X 0,Y 640.772,Z 341.408,A -85,B 0,C 180,E1 30578.583,E2 30578.583} C_VEL
LIN {X 0,Y 640.789,Z 341.403,A -85,B 0,C 180,E1 30575.771,E2 30575.771} C_VEL
LIN {X 0,Y 640.777,Z 341.403,A -85,B 0,C 180,E1 30572.592,E2 30572.592} C_VEL
LIN {X 0,Y 640.771,Z 341.409,A -85,B 0,C 180,E1 30569.94,E2 30569.94} C_VEL
LIN {X 0,Y 640.807,Z 341.409,A -85,B 0,C 180,E1 30566.791,E2 30566.791} C_VEL
LIN {X 0,Y 640.766,Z 341.412,A -85,B 0,C 180,E1 30563.932,E2 30563.932} C_VEL
LIN {X 0,Y 640.826,Z 341.407,A -85,B 0,C 180,E1 30560.848,E2 30560.848} C_VEL
LIN {X 0,Y 640.763,Z 341.411,A -85,B 0,C 180,E1 30557.969,E2 30557.969} C_VEL
LIN {X 0,Y 640.833,Z 341.407,A -85,B 0,C 180,E1 30554.976,E2 30554.976} C_VEL
LIN {X 0,Y 640.837,Z 341.434,A -85,B 0,C 180,E1 30552.923,E2 30552.923} C_VEL
LIN {X 0,Y 648.847,Z 362.263,A -85,B 0,C 180,E1 30550.492,E2 30550.492} C_VEL
LIN {X 0,Y 654.011,Z 376.024,A -85,B 0,C 180,E1 30549.009,E2 30549.009} C_VEL
LIN {X 0,Y 655.595,Z 379.441,A -85,B 0,C 180,E1 30548.85,E2 30548.85} C_VEL
LIN {X 0,Y 661.495,Z 404.617,A -85,B 0,C 180,E1 30548.102,E2 30548.102} C_VEL
LIN {X 0,Y 657.99,Z 671.647,A -85,B 0,C 180,E1 30544.793,E2 30544.793} C_VEL
LIN {X 0,Y 656.699,Z 767.707,A -85,B 0,C 180,E1 30543.599,E2 30543.599} C_VEL
LIN {X 0,Y 655.892,Z 793.05,A -85,B 0,C 180,E1 30543.129,E2 30543.129} C_VEL
LIN {X 0,Y 655.03,Z 813.506,A -85,B 0,C 180,E1 30542.621,E2 30542.621} C_VEL
LIN {X 0,Y 653.952,Z 836.425,A -85,B 0,C 180,E1 30541.914,E2 30541.914} C_VEL
LIN {X 0,Y 652.608,Z 859.258,A -85,B 0,C 180,E1 30541.035,E2 30541.035} C_VEL
LIN {X 0,Y 651.357,Z 880.271,A -85,B 0,C 180,E1 30540.08,E2 30540.08} C_VEL
LIN {X 0,Y 649.815,Z 902.324,A -85,B 0,C 180,E1 30538.891,E2 30538.891} C_VEL
LIN {X 0,Y 648.444,Z 921.455,A -85,B 0,C 180,E1 30537.704,E2 30537.704} C_VEL
LIN {X 0,Y 646.957,Z 941.998,A -85,B 0,C 180,E1 30536.233,E2 30536.233} C_VEL
LIN {X 0,Y 645.698,Z 959.036,A -85,B 0,C 180,E1 30534.845,E2 30534.845} C_VEL
LIN {X 0,Y 644.315,Z 978.602,A -85,B 0,C 180,E1 30533.021,E2 30533.021} C_VEL
LIN {X 0,Y 643.282,Z 993.856,A -85,B 0,C 180,E1 30531.399,E2 30531.399} C_VEL
LIN {X 0,Y 642.297,Z 1009.819,A -85,B 0,C 180,E1 30529.46,E2 30529.46} C_VEL
LIN {X 0,Y 641.577,Z 1022.517,A -85,B 0,C 180,E1 30527.692,E2 30527.692} C_VEL
LIN {X 0,Y 640.946,Z 1035.769,A -85,B 0,C 180,E1 30525.565,E2 30525.565} C_VEL
LIN {X 0,Y 640.557,Z 1045.561,A -85,B 0,C 180,E1 30523.725,E2 30523.725} C_VEL
LIN {X 0,Y 640.244,Z 1055.479,A -85,B 0,C 180,E1 30521.531,E2 30521.531} C_VEL
LIN {X 0,Y 640.064,Z 1062.514,A -85,B 0,C 180,E1 30519.622,E2 30519.622} C_VEL
LIN {X 0,Y 639.958,Z 1068.507,A -85,B 0,C 180,E1 30517.632,E2 30517.632} C_VEL
LIN {X 0,Y 639.926,Z 1073.336,A -85,B 0,C 180,E1 30515.469,E2 30515.469} C_VEL
LIN {X 0,Y 639.908,Z 1076.238,A -85,B 0,C 180,E1 30513.583,E2 30513.583} C_VEL
LIN {X 0,Y 639.894,Z 1078.146,A -85,B 0,C 180,E1 30511.433,E2 30511.433} C_VEL
LIN {X 0,Y 639.894,Z 1078.35,A -85,B 0,C 180,E1 30509.373,E2 30509.373} C_VEL
LIN {X 0,Y 639.907,Z 1077.293,A -85,B 0,C 180,E1 30507.403,E2 30507.403} C_VEL
LIN {X 0,Y 639.924,Z 1074.451,A -85,B 0,C 180,E1 30505.16,E2 30505.16} C_VEL
LIN {X 0,Y 639.935,Z 1070.689,A -85,B 0,C 180,E1 30503.27,E2 30503.27} C_VEL
LIN {X 0,Y 640.008,Z 1065.202,A -85,B 0,C 180,E1 30501.193,E2 30501.193} C_VEL
LIN {X 0,Y 640.169,Z 1057.956,A -85,B 0,C 180,E1 30499.106,E2 30499.106} C_VEL
LIN {X 0,Y 640.404,Z 1049.938,A -85,B 0,C 180,E1 30497.19,E2 30497.19} C_VEL
LIN {X 0,Y 640.813,Z 1038.847,A -85,B 0,C 180,E1 30494.985,E2 30494.985} C_VEL
LIN {X 0,Y 641.3,Z 1027.973,A -85,B 0,C 180,E1 30493.142,E2 30493.142} C_VEL
LIN {X 0,Y 642.038,Z 1014.022,A -85,B 0,C 180,E1 30491.099,E2 30491.099} C_VEL
LIN {X 0,Y 642.841,Z 1000.849,A -85,B 0,C 180,E1 30489.419,E2 30489.419} C_VEL
LIN {X 0,Y 643.933,Z 984.157,A -85,B 0,C 180,E1 30487.543,E2 30487.543} C_VEL
LIN {X 0,Y 645.033,Z 968.318,A -85,B 0,C 180,E1 30485.989,E2 30485.989} C_VEL
LIN {X 0,Y 646.361,Z 950.193,A -85,B 0,C 180,E1 30484.406,E2 30484.406} C_VEL
LIN {X 0,Y 647.746,Z 931.053,A -85,B 0,C 180,E1 30482.96,E2 30482.96} C_VEL
LIN {X 0,Y 649.228,Z 911.161,A -85,B 0,C 180,E1 30481.632,E2 30481.632} C_VEL
LIN {X 0,Y 650.632,Z 890.298,A -85,B 0,C 180,E1 30480.439,E2 30480.439} C_VEL
LIN {X 0,Y 651.972,Z 870.217,A -85,B 0,C 180,E1 30479.443,E2 30479.443} C_VEL
LIN {X 0,Y 653.351,Z 847.074,A -85,B 0,C 180,E1 30478.478,E2 30478.478} C_VEL
LIN {X 0,Y 654.406,Z 826.841,A -85,B 0,C 180,E1 30477.775,E2 30477.775} C_VEL
LIN {X 0,Y 655.479,Z 803.653,A -85,B 0,C 180,E1 30477.111,E2 30477.111} C_VEL
LIN {X 0,Y 656.328,Z 779.728,A -85,B 0,C 180,E1 30476.603,E2 30476.603} C_VEL
LIN {X 0,Y 656.97,Z 755.117,A -85,B 0,C 180,E1 30476.225,E2 30476.225} C_VEL
LIN {X 0,Y 660.095,Z 506.842,A -85,B 0,C 180,E1 30473.173,E2 30473.173} C_VEL
LIN {X 0,Y 661.336,Z 403.158,A -85,B 0,C 180,E1 30471.867,E2 30471.867} C_VEL
LIN {X 0,Y 655.032,Z 377.89,A -85,B 0,C 180,E1 30471.089,E2 30471.089} C_VEL
LIN {X 0,Y 653.661,Z 375.262,A -85,B 0,C 180,E1 30470.933,E2 30470.933} C_VEL
LIN {X 0,Y 645.884,Z 354.531,A -85,B 0,C 180,E1 30468.662,E2 30468.662} C_VEL
LIN {X 0,Y 640.832,Z 341.411,A -85,B 0,C 180,E1 30467.134,E2 30467.134} C_VEL
LIN {X 0,Y 640.763,Z 341.414,A -85,B 0,C 180,E1 30464.105,E2 30464.105} C_VEL
LIN {X 0,Y 640.837,Z 341.408,A -85,B 0,C 180,E1 30461.095,E2 30461.095} C_VEL
LIN {X 0,Y 640.764,Z 341.409,A -85,B 0,C 180,E1 30458.053,E2 30458.053} C_VEL
LIN {X 0,Y 640.817,Z 341.408,A -85,B 0,C 180,E1 30455.153,E2 30455.153} C_VEL
LIN {X 0,Y 640.766,Z 341.408,A -85,B 0,C 180,E1 30452.043,E2 30452.043} C_VEL
LIN {X 0,Y 640.795,Z 341.406,A -85,B 0,C 180,E1 30449.236,E2 30449.236} C_VEL
LIN {X 0,Y 640.777,Z 341.41,A -85,B 0,C 180,E1 30446.107,E2 30446.107} C_VEL
LIN {X 0,Y 640.777,Z 341.397,A -85,B 0,C 180,E1 30443.35,E2 30443.35} C_VEL
LIN {X 0,Y 640.782,Z 341.403,A -85,B 0,C 180,E1 30440.078,E2 30440.078} C_VEL
LIN {X 0,Y 640.777,Z 341.406,A -85,B 0,C 180,E1 30437.247,E2 30437.247} C_VEL
LIN {X 0,Y 640.784,Z 341.403,A -85,B 0,C 180,E1 30433.997,E2 30433.997} C_VEL
LIN {X 0,Y 640.77,Z 341.407,A -85,B 0,C 180,E1 30431.248,E2 30431.248} C_VEL
LIN {X 0,Y 640.804,Z 341.408,A -85,B 0,C 180,E1 30428.073,E2 30428.073} C_VEL
LIN {X 0,Y 640.766,Z 341.401,A -85,B 0,C 180,E1 30425.283,E2 30425.283} C_VEL
LIN {X 0,Y 640.831,Z 341.407,A -85,B 0,C 180,E1 30422.236,E2 30422.236} C_VEL
LIN {X 0,Y 640.763,Z 341.394,A -85,B 0,C 180,E1 30419.285,E2 30419.285} C_VEL
LIN {X 0,Y 640.831,Z 341.406,A -85,B 0,C 180,E1 30416.332,E2 30416.332} C_VEL
LIN {X 0,Y 640.765,Z 341.403,A -85,B 0,C 180,E1 30413.279,E2 30413.279} C_VEL
LIN {X 0,Y 640.819,Z 341.405,A -85,B 0,C 180,E1 30410.389,E2 30410.389} C_VEL
LIN {X 0,Y 640.771,Z 341.409,A -85,B 0,C 180,E1 30407.29,E2 30407.29} C_VEL
LIN {X 0,Y 640.792,Z 341.402,A -85,B 0,C 180,E1 30404.524,E2 30404.524} C_VEL
LIN {X 0,Y 640.78,Z 341.41,A -85,B 0,C 180,E1 30401.344,E2 30401.344} C_VEL
LIN {X 0,Y 640.779,Z 341.397,A -85,B 0,C 180,E1 30398.584,E2 30398.584} C_VEL
LIN {X 0,Y 640.79,Z 341.4,A -85,B 0,C 180,E1 30395.378,E2 30395.378} C_VEL
LIN {X 0,Y 640.775,Z 341.408,A -85,B 0,C 180,E1 30392.591,E2 30392.591} C_VEL
LIN {X 0,Y 640.814,Z 341.405,A -85,B 0,C 180,E1 30389.464,E2 30389.464} C_VEL
LIN {X 0,Y 640.769,Z 341.4,A -85,B 0,C 180,E1 30386.575,E2 30386.575} C_VEL
LIN {X 0,Y 640.823,Z 341.401,A -85,B 0,C 180,E1 30383.472,E2 30383.472} C_VEL
LIN {X 0,Y 640.767,Z 341.406,A -85,B 0,C 180,E1 30380.572,E2 30380.572} C_VEL
LIN {X 0,Y 640.834,Z 341.399,A -85,B 0,C 180,E1 30377.563,E2 30377.563} C_VEL
LIN {X 0,Y 640.768,Z 341.396,A -85,B 0,C 180,E1 30374.604,E2 30374.604} C_VEL
LIN {X 0,Y 640.768,Z 341.399,A -85,B 0,C 180,E1 30374.487,E2 30374.487} C_VEL
LIN {X 0,Y 639.803,Z 341.532,A -85,B 0,C 180,E1 30373.799,E2 30373.799} C_VEL
LIN {X 0,Y 633.446,Z 342.32,A -85,B 0,C 180,E1 30371.867,E2 30371.867} C_VEL
LIN {X 0,Y 632.899,Z 342.393,A -85,B 0,C 180,E1 30371.365,E2 30371.365} C_VEL
LIN {X 0,Y 632.911,Z 342.613,A -85,B 0,C 180,E1 30369.161,E2 30369.161} C_VEL
LIN {X 0,Y 635.679,Z 349.892,A -85,B 0,C 180,E1 30368.288,E2 30368.288} C_VEL
LIN {X 0,Y 653.275,Z 378.692,A -85,B 0,C 180,E1 30366.602,E2 30366.602} C_VEL
LIN {X 0,Y 655.217,Z 382.638,A -85,B 0,C 180,E1 30366.412,E2 30366.412} C_VEL
LIN {X 0,Y 651.805,Z 620.683,A -85,B 0,C 180,E1 30363.423,E2 30363.423} C_VEL
LIN {X 0,Y 650.1,Z 738.3,A -85,B 0,C 180,E1 30361.947,E2 30361.947} C_VEL
LIN {X 0,Y 649.255,Z 763.745,A -85,B 0,C 180,E1 30361.472,E2 30361.472} C_VEL
LIN {X 0,Y 648.345,Z 784.012,A -85,B 0,C 180,E1 30360.963,E2 30360.963} C_VEL
LIN {X 0,Y 647.226,Z 806.04,A -85,B 0,C 180,E1 30360.277,E2 30360.277} C_VEL
LIN {X 0,Y 645.756,Z 828.772,A -85,B 0,C 180,E1 30359.396,E2 30359.396} C_VEL
LIN {X 0,Y 644.399,Z 849.399,A -85,B 0,C 180,E1 30358.448,E2 30358.448} C_VEL
LIN {X 0,Y 642.764,Z 871.198,A -85,B 0,C 180,E1 30357.266,E2 30357.266} C_VEL
LIN {X 0,Y 641.223,Z 890.882,A -85,B 0,C 180,E1 30356.037,E2 30356.037} C_VEL
LIN {X 0,Y 639.565,Z 912.066,A -85,B 0,C 180,E1 30354.509,E2 30354.509} C_VEL
LIN {X 0,Y 638.248,Z 928.795,A -85,B 0,C 180,E1 30353.131,E2 30353.131} C_VEL
LIN {X 0,Y 636.792,Z 947.66,A -85,B 0,C 180,E1 30351.364,E2 30351.364} C_VEL
LIN {X 0,Y 635.693,Z 962.6,A -85,B 0,C 180,E1 30349.766,E2 30349.766} C_VEL
LIN {X 0,Y 634.597,Z 978.807,A -85,B 0,C 180,E1 30347.799,E2 30347.799} C_VEL
LIN {X 0,Y 633.792,Z 991.484,A -85,B 0,C 180,E1 30346.027,E2 30346.027} C_VEL
LIN {X 0,Y 633.129,Z 1004.305,A -85,B 0,C 180,E1 30343.983,E2 30343.983} C_VEL
LIN {X 0,Y 632.653,Z 1014.647,A -85,B 0,C 180,E1 30342.042,E2 30342.042} C_VEL
LIN {X 0,Y 632.324,Z 1023.928,A -85,B 0,C 180,E1 30340.017,E2 30340.017} C_VEL
LIN {X 0,Y 632.091,Z 1031.819,A -85,B 0,C 180,E1 30337.91,E2 30337.91} C_VEL
LIN {X 0,Y 631.988,Z 1037.646,A -85,B 0,C 180,E1 30335.994,E2 30335.994} C_VEL
LIN {X 0,Y 631.929,Z 1042.939,A -85,B 0,C 180,E1 30333.72,E2 30333.72} C_VEL
LIN {X 0,Y 631.914,Z 1046.063,A -85,B 0,C 180,E1 30331.723,E2 30331.723} C_VEL
LIN {X 0,Y 631.902,Z 1047.932,A -85,B 0,C 180,E1 30329.728,E2 30329.728} C_VEL
LIN {X 0,Y 631.893,Z 1048.385,A -85,B 0,C 180,E1 30327.461,E2 30327.461} C_VEL
LIN {X 0,Y 631.905,Z 1047.464,A -85,B 0,C 180,E1 30325.553,E2 30325.553} C_VEL
LIN {X 0,Y 631.923,Z 1044.999,A -85,B 0,C 180,E1 30323.367,E2 30323.367} C_VEL
LIN {X 0,Y 631.944,Z 1040.969,A -85,B 0,C 180,E1 30321.263,E2 30321.263} C_VEL
LIN {X 0,Y 632.006,Z 1036.026,A -85,B 0,C 180,E1 30319.333,E2 30319.333} C_VEL
LIN {X 0,Y 632.182,Z 1028.337,A -85,B 0,C 180,E1 30317.021,E2 30317.021} C_VEL
LIN {X 0,Y 632.43,Z 1020.718,A -85,B 0,C 180,E1 30315.16,E2 30315.16} C_VEL
LIN {X 0,Y 632.854,Z 1010.256,A -85,B 0,C 180,E1 30313.005,E2 30313.005} C_VEL
LIN {X 0,Y 633.396,Z 998.832,A -85,B 0,C 180,E1 30311.023,E2 30311.023} C_VEL
LIN {X 0,Y 634.177,Z 985.19,A -85,B 0,C 180,E1 30308.97,E2 30308.97} C_VEL
LIN {X 0,Y 635.064,Z 971.658,A -85,B 0,C 180,E1 30307.212,E2 30307.212} C_VEL
LIN {X 0,Y 636.229,Z 955.363,A -85,B 0,C 180,E1 30305.338,E2 30305.338} C_VEL
LIN {X 0,Y 637.495,Z 938.385,A -85,B 0,C 180,E1 30303.649,E2 30303.649} C_VEL
LIN {X 0,Y 638.921,Z 920.3,A -85,B 0,C 180,E1 30302.05,E2 30302.05} C_VEL
LIN {X 0,Y 640.414,Z 901.338,A -85,B 0,C 180,E1 30300.601,E2 30300.601} C_VEL
LIN {X 0,Y 641.967,Z 881.759,A -85,B 0,C 180,E1 30299.278,E2 30299.278} C_VEL
LIN {X 0,Y 643.591,Z 859.914,A -85,B 0,C 180,E1 30298.009,E2 30298.009} C_VEL
LIN {X 0,Y 645.086,Z 839.544,A -85,B 0,C 180,E1 30296.988,E2 30296.988} C_VEL
LIN {X 0,Y 646.555,Z 816.902,A -85,B 0,C 180,E1 30296.036,E2 30296.036} C_VEL
LIN {X 0,Y 647.698,Z 796.749,A -85,B 0,C 180,E1 30295.328,E2 30295.328} C_VEL
LIN {X 0,Y 648.85,Z 773.049,A -85,B 0,C 180,E1 30294.651,E2 30294.651} C_VEL
LIN {X 0,Y 649.724,Z 750.211,A -85,B 0,C 180,E1 30294.164,E2 30294.164} C_VEL
LIN {X 0,Y 650.389,Z 725.478,A -85,B 0,C 180,E1 30293.782,E2 30293.782} C_VEL
LIN {X 0,Y 653.922,Z 472.185,A -85,B 0,C 180,E1 30290.632,E2 30290.632} C_VEL
LIN {X 0,Y 655.065,Z 381.929,A -85,B 0,C 180,E1 30289.478,E2 30289.478} C_VEL
LIN {X 0,Y 644.365,Z 363.809,A -85,B 0,C 180,E1 30288.446,E2 30288.446} C_VEL
LIN {X 0,Y 635.544,Z 349.449,A -85,B 0,C 180,E1 30287.551,E2 30287.551} C_VEL
LIN {X 0,Y 632.89,Z 342.397,A -85,B 0,C 180,E1 30286.625,E2 30286.625} C_VEL
LIN {X 0,Y 632.83,Z 342.395,A -85,B 0,C 180,E1 30283.543,E2 30283.543} C_VEL
LIN {X 0,Y 632.893,Z 342.367,A -85,B 0,C 180,E1 30280.543,E2 30280.543} C_VEL
LIN {X 0,Y 632.83,Z 342.398,A -85,B 0,C 180,E1 30277.468,E2 30277.468} C_VEL
LIN {X 0,Y 632.876,Z 342.376,A -85,B 0,C 180,E1 30274.555,E2 30274.555} C_VEL
LIN {X 0,Y 632.831,Z 342.39,A -85,B 0,C 180,E1 30271.427,E2 30271.427} C_VEL
LIN {X 0,Y 632.86,Z 342.394,A -85,B 0,C 180,E1 30268.602,E2 30268.602} C_VEL
LIN {X 0,Y 632.837,Z 342.39,A -85,B 0,C 180,E1 30265.453,E2 30265.453} C_VEL
LIN {X 0,Y 632.843,Z 342.401,A -85,B 0,C 180,E1 30262.673,E2 30262.673} C_VEL
LIN {X 0,Y 632.841,Z 342.396,A -85,B 0,C 180,E1 30259.378,E2 30259.378} C_VEL
LIN {X 0,Y 632.847,Z 342.396,A -85,B 0,C 180,E1 30256.523,E2 30256.523} C_VEL
LIN {X 0,Y 632.839,Z 342.393,A -85,B 0,C 180,E1 30253.274,E2 30253.274} C_VEL
LIN {X 0,Y 632.842,Z 342.397,A -85,B 0,C 180,E1 30250.469,E2 30250.469} C_VEL
LIN {X 0,Y 632.846,Z 342.395,A -85,B 0,C 180,E1 30247.262,E2 30247.262} C_VEL
LIN {X 0,Y 632.836,Z 342.394,A -85,B 0,C 180,E1 30244.44,E2 30244.44} C_VEL
LIN {X 0,Y 632.856,Z 342.388,A -85,B 0,C 180,E1 30241.267,E2 30241.267} C_VEL
LIN {X 0,Y 632.83,Z 342.399,A -85,B 0,C 180,E1 30238.461,E2 30238.461} C_VEL
LIN {X 0,Y 632.88,Z 342.396,A -85,B 0,C 180,E1 30235.378,E2 30235.378} C_VEL
LIN {X 0,Y 632.824,Z 342.387,A -85,B 0,C 180,E1 30232.464,E2 30232.464} C_VEL
LIN {X 0,Y 632.891,Z 342.385,A -85,B 0,C 180,E1 30229.44,E2 30229.44} C_VEL
LIN {X 0,Y 632.825,Z 342.398,A -85,B 0,C 180,E1 30226.476,E2 30226.476} C_VEL
LIN {X 0,Y 632.893,Z 342.391,A -85,B 0,C 180,E1 30223.478,E2 30223.478} C_VEL
LIN {X 0,Y 632.823,Z 342.386,A -85,B 0,C 180,E1 30220.429,E2 30220.429} C_VEL
LIN {X 0,Y 632.9,Z 342.387,A -85,B 0,C 180,E1 30217.424,E2 30217.424} C_VEL
LIN {X 0,Y 632.825,Z 342.398,A -85,B 0,C 180,E1 30214.346,E2 30214.346} C_VEL
LIN {X 0,Y 632.888,Z 342.398,A -85,B 0,C 180,E1 30211.399,E2 30211.399} C_VEL
LIN {X 0,Y 632.827,Z 342.398,A -85,B 0,C 180,E1 30208.36,E2 30208.36} C_VEL
LIN {X 0,Y 632.855,Z 342.402,A -85,B 0,C 180,E1 30205.554,E2 30205.554} C_VEL
LIN {X 0,Y 632.837,Z 342.397,A -85,B 0,C 180,E1 30202.419,E2 30202.419} C_VEL
LIN {X 0,Y 632.84,Z 342.403,A -85,B 0,C 180,E1 30199.624,E2 30199.624} C_VEL
LIN {X 0,Y 632.839,Z 342.399,A -85,B 0,C 180,E1 30196.333,E2 30196.333} C_VEL
LIN {X 0,Y 632.852,Z 342.489,A -85,B 0,C 180,E1 30193.494,E2 30193.494} C_VEL
LIN {X 0,Y 641.382,Z 364.278,A -85,B 0,C 180,E1 30190.878,E2 30190.878} C_VEL
LIN {X 0,Y 645.735,Z 375.741,A -85,B 0,C 180,E1 30189.614,E2 30189.614} C_VEL
LIN {X 0,Y 649.816,Z 383.299,A -85,B 0,C 180,E1 30189.209,E2 30189.209} C_VEL
LIN {X 0,Y 655.154,Z 406.516,A -85,B 0,C 180,E1 30188.509,E2 30188.509} C_VEL
LIN {X 0,Y 651.364,Z 674.738,A -85,B 0,C 180,E1 30185.155,E2 30185.155} C_VEL
LIN {X 0,Y 650.015,Z 767.474,A -85,B 0,C 180,E1 30183.991,E2 30183.991} C_VEL
LIN {X 0,Y 649.153,Z 792.825,A -85,B 0,C 180,E1 30183.518,E2 30183.518} C_VEL
LIN {X 0,Y 648.242,Z 813.064,A -85,B 0,C 180,E1 30183.013,E2 30183.013} C_VEL
LIN {X 0,Y 647.093,Z 835.946,A -85,B 0,C 180,E1 30182.303,E2 30182.303} C_VEL
LIN {X 0,Y 645.644,Z 858.657,A -85,B 0,C 180,E1 30181.425,E2 30181.425} C_VEL
LIN {X 0,Y 644.282,Z 880.095,A -85,B 0,C 180,E1 30180.445,E2 30180.445} C_VEL
LIN {X 0,Y 642.66,Z 902.269,A -85,B 0,C 180,E1 30179.245,E2 30179.245} C_VEL
LIN {X 0,Y 641.294,Z 919.982,A -85,B 0,C 180,E1 30178.141,E2 30178.141} C_VEL
LIN {X 0,Y 639.606,Z 941.565,A -85,B 0,C 180,E1 30176.593,E2 30176.593} C_VEL
LIN {X 0,Y 638.282,Z 958.285,A -85,B 0,C 180,E1 30175.22,E2 30175.22} C_VEL
LIN {X 0,Y 636.866,Z 976.749,A -85,B 0,C 180,E1 30173.502,E2 30173.502} C_VEL
LIN {X 0,Y 635.732,Z 991.986,A -85,B 0,C 180,E1 30171.88,E2 30171.88} C_VEL
LIN {X 0,Y 634.663,Z 1007.703,A -85,B 0,C 180,E1 30169.991,E2 30169.991} C_VEL
LIN {X 0,Y 633.812,Z 1021.246,A -85,B 0,C 180,E1 30168.106,E2 30168.106} C_VEL
LIN {X 0,Y 633.141,Z 1034.211,A -85,B 0,C 180,E1 30166.044,E2 30166.044} C_VEL
LIN {X 0,Y 632.653,Z 1044.642,A -85,B 0,C 180,E1 30164.087,E2 30164.087} C_VEL
LIN {X 0,Y 632.316,Z 1053.991,A -85,B 0,C 180,E1 30162.048,E2 30162.048} C_VEL
LIN {X 0,Y 632.086,Z 1061.907,A -85,B 0,C 180,E1 30159.929,E2 30159.929} C_VEL
LIN {X 0,Y 631.983,Z 1067.745,A -85,B 0,C 180,E1 30158.003,E2 30158.003} C_VEL
LIN {X 0,Y 631.933,Z 1073.016,A -85,B 0,C 180,E1 30155.721,E2 30155.721} C_VEL
LIN {X 0,Y 631.906,Z 1076.124,A -85,B 0,C 180,E1 30153.72,E2 30153.72} C_VEL
LIN {X 0,Y 631.896,Z 1077.969,A -85,B 0,C 180,E1 30151.723,E2 30151.723} C_VEL
LIN {X 0,Y 631.893,Z 1078.395,A -85,B 0,C 180,E1 30149.547,E2 30149.547} C_VEL
LIN {X 0,Y 631.909,Z 1077.428,A -85,B 0,C 180,E1 30147.551,E2 30147.551} C_VEL
LIN {X 0,Y 631.922,Z 1074.768,A -85,B 0,C 180,E1 30145.28,E2 30145.28} C_VEL
LIN {X 0,Y 631.937,Z 1070.896,A -85,B 0,C 180,E1 30143.276,E2 30143.276} C_VEL
LIN {X 0,Y 632.01,Z 1065.71,A -85,B 0,C 180,E1 30141.264,E2 30141.264} C_VEL
LIN {X 0,Y 632.188,Z 1058.309,A -85,B 0,C 180,E1 30139.059,E2 30139.059} C_VEL
LIN {X 0,Y 632.439,Z 1050.346,A -85,B 0,C 180,E1 30137.119,E2 30137.119} C_VEL
LIN {X 0,Y 632.886,Z 1039.247,A -85,B 0,C 180,E1 30134.866,E2 30134.866} C_VEL
LIN {X 0,Y 633.408,Z 1028.544,A -85,B 0,C 180,E1 30133.02,E2 30133.02} C_VEL
LIN {X 0,Y 634.203,Z 1014.721,A -85,B 0,C 180,E1 30130.952,E2 30130.952} C_VEL
LIN {X 0,Y 635.122,Z 1000.847,A -85,B 0,C 180,E1 30129.158,E2 30129.158} C_VEL
LIN {X 0,Y 636.308,Z 984.156,A -85,B 0,C 180,E1 30127.259,E2 30127.259} C_VEL
LIN {X 0,Y 637.505,Z 968.256,A -85,B 0,C 180,E1 30125.681,E2 30125.681} C_VEL
LIN {X 0,Y 638.959,Z 949.758,A -85,B 0,C 180,E1 30124.052,E2 30124.052} C_VEL
LIN {X 0,Y 640.432,Z 931.059,A -85,B 0,C 180,E1 30122.626,E2 30122.626} C_VEL
LIN {X 0,Y 642.048,Z 910.744,A -85,B 0,C 180,E1 30121.258,E2 30121.258} C_VEL
LIN {X 0,Y 643.519,Z 890.231,A -85,B 0,C 180,E1 30120.082,E2 30120.082} C_VEL
LIN {X 0,Y 644.949,Z 869.999,A -85,B 0,C 180,E1 30119.074,E2 30119.074} C_VEL
LIN {X 0,Y 646.408,Z 847.179,A -85,B 0,C 180,E1 30118.113,E2 30118.113} C_VEL
LIN {X 0,Y 647.553,Z 826.623,A -85,B 0,C 180,E1 30117.392,E2 30117.392} C_VEL
LIN {X 0,Y 648.715,Z 803.161,A -85,B 0,C 180,E1 30116.717,E2 30116.717} C_VEL
LIN {X 0,Y 649.634,Z 779.407,A -85,B 0,C 180,E1 30116.211,E2 30116.211} C_VEL
LIN {X 0,Y 650.311,Z 754.76,A -85,B 0,C 180,E1 30115.83,E2 30115.83} C_VEL
LIN {X 0,Y 653.692,Z 505.738,A -85,B 0,C 180,E1 30112.74,E2 30112.74} C_VEL
LIN {X 0,Y 654.989,Z 404.942,A -85,B 0,C 180,E1 30111.458,E2 30111.458} C_VEL
LIN {X 0,Y 649.257,Z 381.898,A -85,B 0,C 180,E1 30110.738,E2 30110.738} C_VEL
LIN {X 0,Y 645.352,Z 374.901,A -85,B 0,C 180,E1 30110.332,E2 30110.332} C_VEL
LIN {X 0,Y 637.667,Z 355.005,A -85,B 0,C 180,E1 30108.088,E2 30108.088} C_VEL
LIN {X 0,Y 632.849,Z 342.404,A -85,B 0,C 180,E1 30106.584,E2 30106.584} C_VEL
LIN {X 0,Y 632.833,Z 342.402,A -85,B 0,C 180,E1 30103.774,E2 30103.774} C_VEL
LIN {X 0,Y 632.861,Z 342.395,A -85,B 0,C 180,E1 30100.613,E2 30100.613} C_VEL
LIN {X 0,Y 632.826,Z 342.397,A -85,B 0,C 180,E1 30097.811,E2 30097.811} C_VEL
LIN {X 0,Y 632.888,Z 342.39,A -85,B 0,C 180,E1 30094.761,E2 30094.761} C_VEL
LIN {X 0,Y 632.824,Z 342.395,A -85,B 0,C 180,E1 30091.781,E2 30091.781} C_VEL
LIN {X 0,Y 632.902,Z 342.395,A -85,B 0,C 180,E1 30088.739,E2 30088.739} C_VEL
LIN {X 0,Y 632.826,Z 342.398,A -85,B 0,C 180,E1 30085.754,E2 30085.754} C_VEL
LIN {X 0,Y 632.896,Z 342.382,A -85,B 0,C 180,E1 30082.772,E2 30082.772} C_VEL
LIN {X 0,Y 632.825,Z 342.391,A -85,B 0,C 180,E1 30079.763,E2 30079.763} C_VEL
LIN {X 0,Y 632.882,Z 342.394,A -85,B 0,C 180,E1 30076.805,E2 30076.805} C_VEL
LIN {X 0,Y 632.828,Z 342.394,A -85,B 0,C 180,E1 30073.71,E2 30073.71} C_VEL
LIN {X 0,Y 632.866,Z 342.395,A -85,B 0,C 180,E1 30070.837,E2 30070.837} C_VEL
LIN {X 0,Y 632.832,Z 342.4,A -85,B 0,C 180,E1 30067.718,E2 30067.718} C_VEL
LIN {X 0,Y 632.849,Z 342.388,A -85,B 0,C 180,E1 30064.894,E2 30064.894} C_VEL
LIN {X 0,Y 632.841,Z 342.399,A -85,B 0,C 180,E1 30061.72,E2 30061.72} C_VEL
LIN {X 0,Y 632.838,Z 342.381,A -85,B 0,C 180,E1 30058.914,E2 30058.914} C_VEL
LIN {X 0,Y 632.844,Z 342.394,A -85,B 0,C 180,E1 30055.65,E2 30055.65} C_VEL
LIN {X 0,Y 632.838,Z 342.39,A -85,B 0,C 180,E1 30052.83,E2 30052.83} C_VEL
LIN {X 0,Y 632.85,Z 342.386,A -85,B 0,C 180,E1 30049.623,E2 30049.623} C_VEL
LIN {X 0,Y 632.84,Z 342.396,A -85,B 0,C 180,E1 30046.726,E2 30046.726} C_VEL
LIN {X 0,Y 632.847,Z 342.39,A -85,B 0,C 180,E1 30043.477,E2 30043.477} C_VEL
LIN {X 0,Y 632.843,Z 342.395,A -85,B 0,C 180,E1 30040.606,E2 30040.606} C_VEL
LIN {X 0,Y 632.846,Z 342.4,A -85,B 0,C 180,E1 30037.324,E2 30037.324} C_VEL
LIN {X 0,Y 632.836,Z 342.384,A -85,B 0,C 180,E1 30034.547,E2 30034.547} C_VEL
LIN {X 0,Y 632.861,Z 342.39,A -85,B 0,C 180,E1 30031.398,E2 30031.398} C_VEL
LIN {X 0,Y 632.834,Z 342.398,A -85,B 0,C 180,E1 30028.562,E2 30028.562} C_VEL
LIN {X 0,Y 632.879,Z 342.396,A -85,B 0,C 180,E1 30025.445,E2 30025.445} C_VEL
LIN {X 0,Y 632.833,Z 342.396,A -85,B 0,C 180,E1 30022.483,E2 30022.483} C_VEL
LIN {X 0,Y 632.887,Z 342.393,A -85,B 0,C 180,E1 30019.389,E2 30019.389} C_VEL
LIN {X 0,Y 632.83,Z 342.374,A -85,B 0,C 180,E1 30016.457,E2 30016.457} C_VEL
LIN {X 0,Y 632.892,Z 342.399,A -85,B 0,C 180,E1 30013.386,E2 30013.386} C_VEL
LIN {X 0,Y 632.899,Z 342.393,A -85,B 0,C 180,E1 30011.365,E2 30011.365} C_VEL
LIN {X 0,Y 631.782,Z 342.539,A -85,B 0,C 180,E1 30010.878,E2 30010.878} C_VEL
LIN {X 0,Y 627.397,Z 343.543,A -85,B 0,C 180,E1 30010.04,E2 30010.04} C_VEL
LIN {X 0,Y 625.956,Z 345.103,A -85,B 0,C 180,E1 30009.601,E2 30009.601} C_VEL
LIN {X 0,Y 626.203,Z 346.794,A -85,B 0,C 180,E1 30009.306,E2 30009.306} C_VEL
LIN {X 0,Y 627.539,Z 350.222,A -85,B 0,C 180,E1 30008.908,E2 30008.908} C_VEL
LIN {X 0,Y 646.136,Z 380.402,A -85,B 0,C 180,E1 30007.085,E2 30007.085} C_VEL
LIN {X 0,Y 648.908,Z 385.733,A -85,B 0,C 180,E1 30006.813,E2 30006.813} C_VEL
LIN {X 0,Y 645.238,Z 625.022,A -85,B 0,C 180,E1 30003.783,E2 30003.783} C_VEL
LIN {X 0,Y 643.473,Z 738.636,A -85,B 0,C 180,E1 30002.344,E2 30002.344} C_VEL
LIN {X 0,Y 642.583,Z 763.969,A -85,B 0,C 180,E1 30001.866,E2 30001.866} C_VEL
LIN {X 0,Y 641.625,Z 784.112,A -85,B 0,C 180,E1 30001.357,E2 30001.357} C_VEL
LIN {X 0,Y 640.412,Z 806.612,A -85,B 0,C 180,E1 30000.65,E2 30000.65} C_VEL
LIN {X 0,Y 638.823,Z 829.621,A -85,B 0,C 180,E1 29999.747,E2 29999.747} C_VEL
LIN {X 0,Y 637.27,Z 851.88,A -85,B 0,C 180,E1 29998.707,E2 29998.707} C_VEL
LIN {X 0,Y 635.566,Z 872.666,A -85,B 0,C 180,E1 29997.55,E2 29997.55} C_VEL
LIN {X 0,Y 633.988,Z 891.348,A -85,B 0,C 180,E1 29996.362,E2 29996.362} C_VEL
LIN {X 0,Y 632.189,Z 912.224,A -85,B 0,C 180,E1 29994.83,E2 29994.83} C_VEL
LIN {X 0,Y 630.789,Z 928.845,A -85,B 0,C 180,E1 29993.445,E2 29993.445} C_VEL
LIN {X 0,Y 629.177,Z 948.129,A -85,B 0,C 180,E1 29991.614,E2 29991.614} C_VEL
LIN {X 0,Y 628.015,Z 962.844,A -85,B 0,C 180,E1 29990.018,E2 29990.018} C_VEL
LIN {X 0,Y 626.82,Z 979.01,A -85,B 0,C 180,E1 29988.027,E2 29988.027} C_VEL
LIN {X 0,Y 625.963,Z 991.667,A -85,B 0,C 180,E1 29986.233,E2 29986.233} C_VEL
LIN {X 0,Y 625.239,Z 1004.457,A -85,B 0,C 180,E1 29984.163,E2 29984.163} C_VEL
LIN {X 0,Y 624.721,Z 1014.778,A -85,B 0,C 180,E1 29982.197,E2 29982.197} C_VEL
LIN {X 0,Y 624.35,Z 1024.445,A -85,B 0,C 180,E1 29980.053,E2 29980.053} C_VEL
LIN {X 0,Y 624.101,Z 1032.207,A -85,B 0,C 180,E1 29977.92,E2 29977.92} C_VEL
LIN {X 0,Y 623.99,Z 1037.972,A -85,B 0,C 180,E1 29975.979,E2 29975.979} C_VEL
LIN {X 0,Y 623.927,Z 1043.144,A -85,B 0,C 180,E1 29973.675,E2 29973.675} C_VEL
LIN {X 0,Y 623.914,Z 1046.095,A -85,B 0,C 180,E1 29971.745,E2 29971.745} C_VEL
LIN {X 0,Y 623.9,Z 1048.018,A -85,B 0,C 180,E1 29969.633,E2 29969.633} C_VEL
LIN {X 0,Y 623.893,Z 1048.378,A -85,B 0,C 180,E1 29967.428,E2 29967.428} C_VEL
LIN {X 0,Y 623.903,Z 1047.444,A -85,B 0,C 180,E1 29965.496,E2 29965.496} C_VEL
LIN {X 0,Y 623.921,Z 1044.954,A -85,B 0,C 180,E1 29963.282,E2 29963.282} C_VEL
LIN {X 0,Y 623.947,Z 1041.117,A -85,B 0,C 180,E1 29961.243,E2 29961.243} C_VEL
LIN {X 0,Y 624.013,Z 1036.208,A -85,B 0,C 180,E1 29959.288,E2 29959.288} C_VEL
LIN {X 0,Y 624.202,Z 1028.589,A -85,B 0,C 180,E1 29956.946,E2 29956.946} C_VEL
LIN {X 0,Y 624.469,Z 1021.007,A -85,B 0,C 180,E1 29955.061,E2 29955.061} C_VEL
LIN {X 0,Y 624.907,Z 1011.141,A -85,B 0,C 180,E1 29952.974,E2 29952.974} C_VEL
LIN {X 0,Y 625.479,Z 999.818,A -85,B 0,C 180,E1 29950.967,E2 29950.967} C_VEL
LIN {X 0,Y 626.249,Z 987.436,A -85,B 0,C 180,E1 29949.044,E2 29949.044} C_VEL
LIN {X 0,Y 627.252,Z 972.986,A -85,B 0,C 180,E1 29947.11,E2 29947.11} C_VEL
LIN {X 0,Y 628.31,Z 959.029,A -85,B 0,C 180,E1 29945.458,E2 29945.458} C_VEL
LIN {X 0,Y 629.781,Z 940.775,A -85,B 0,C 180,E1 29943.567,E2 29943.567} C_VEL
LIN {X 0,Y 631.144,Z 924.5,A -85,B 0,C 180,E1 29942.086,E2 29942.086} C_VEL
LIN {X 0,Y 632.941,Z 903.55,A -85,B 0,C 180,E1 29940.418,E2 29940.418} C_VEL
LIN {X 0,Y 634.459,Z 885.961,A -85,B 0,C 180,E1 29939.19,E2 29939.19} C_VEL
LIN {X 0,Y 636.216,Z 864.814,A -85,B 0,C 180,E1 29937.899,E2 29937.899} C_VEL
LIN {X 0,Y 637.795,Z 844.222,A -85,B 0,C 180,E1 29936.829,E2 29936.829} C_VEL
LIN {X 0,Y 639.412,Z 822.204,A -85,B 0,C 180,E1 29935.848,E2 29935.848} C_VEL
LIN {X 0,Y 640.78,Z 799.713,A -85,B 0,C 180,E1 29935.031,E2 29935.031} C_VEL
LIN {X 0,Y 641.872,Z 779.385,A -85,B 0,C 180,E1 29934.421,E2 29934.421} C_VEL
LIN {X 0,Y 642.964,Z 753.407,A -85,B 0,C 180,E1 29933.822,E2 29933.822} C_VEL
LIN {X 0,Y 643.64,Z 731.33,A -85,B 0,C 180,E1 29933.461,E2 29933.461} C_VEL
LIN {X 0,Y 647.419,Z 481.974,A -85,B 0,C 180,E1 29930.324,E2 29930.324} C_VEL
LIN {X 0,Y 648.81,Z 385.091,A -85,B 0,C 180,E1 29929.076,E2 29929.076} C_VEL
LIN {X 0,Y 635.612,Z 362.835,A -85,B 0,C 180,E1 29927.761,E2 29927.761} C_VEL
LIN {X 0,Y 627.277,Z 349.758,A -85,B 0,C 180,E1 29926.892,E2 29926.892} C_VEL
LIN {X 0,Y 624.924,Z 343.385,A -85,B 0,C 180,E1 29926.056,E2 29926.056} C_VEL
LIN {X 0,Y 624.899,Z 343.386,A -85,B 0,C 180,E1 29923.144,E2 29923.144} C_VEL
LIN {X 0,Y 624.916,Z 343.365,A -85,B 0,C 180,E1 29919.913,E2 29919.913} C_VEL
LIN {X 0,Y 624.894,Z 343.377,A -85,B 0,C 180,E1 29917.102,E2 29917.102} C_VEL
LIN {X 0,Y 624.935,Z 343.381,A -85,B 0,C 180,E1 29913.945,E2 29913.945} C_VEL
LIN {X 0,Y 624.893,Z 343.381,A -85,B 0,C 180,E1 29911.013,E2 29911.013} C_VEL
LIN {X 0,Y 624.949,Z 343.381,A -85,B 0,C 180,E1 29907.956,E2 29907.956} C_VEL
LIN {X 0,Y 624.891,Z 343.38,A -85,B 0,C 180,E1 29904.988,E2 29904.988} C_VEL
LIN {X 0,Y 624.949,Z 343.374,A -85,B 0,C 180,E1 29901.879,E2 29901.879} C_VEL
LIN {X 0,Y 624.89,Z 343.387,A -85,B 0,C 180,E1 29898.955,E2 29898.955} C_VEL
LIN {X 0,Y 624.958,Z 343.383,A -85,B 0,C 180,E1 29895.878,E2 29895.878} C_VEL
LIN {X 0,Y 624.888,Z 343.383,A -85,B 0,C 180,E1 29892.945,E2 29892.945} C_VEL
LIN {X 0,Y 624.952,Z 343.375,A -85,B 0,C 180,E1 29889.95,E2 29889.95} C_VEL
LIN {X 0,Y 624.889,Z 343.385,A -85,B 0,C 180,E1 29886.893,E2 29886.893} C_VEL
LIN {X 0,Y 624.952,Z 343.388,A -85,B 0,C 180,E1 29883.853,E2 29883.853} C_VEL
LIN {X 0,Y 624.887,Z 343.379,A -85,B 0,C 180,E1 29880.825,E2 29880.825} C_VEL
LIN {X 0,Y 624.942,Z 343.379,A -85,B 0,C 180,E1 29877.891,E2 29877.891} C_VEL
LIN {X 0,Y 624.89,Z 343.387,A -85,B 0,C 180,E1 29874.767,E2 29874.767} C_VEL
LIN {X 0,Y 624.926,Z 343.378,A -85,B 0,C 180,E1 29871.906,E2 29871.906} C_VEL
LIN {X 0,Y 624.891,Z 343.374,A -85,B 0,C 180,E1 29868.743,E2 29868.743} C_VEL
LIN {X 0,Y 624.924,Z 343.388,A -85,B 0,C 180,E1 29865.83,E2 29865.83} C_VEL
LIN {X 0,Y 624.895,Z 343.386,A -85,B 0,C 180,E1 29862.685,E2 29862.685} C_VEL
LIN {X 0,Y 624.916,Z 343.377,A -85,B 0,C 180,E1 29859.781,E2 29859.781} C_VEL
LIN {X 0,Y 624.896,Z 343.376,A -85,B 0,C 180,E1 29856.62,E2 29856.62} C_VEL
LIN {X 0,Y 624.908,Z 343.387,A -85,B 0,C 180,E1 29853.793,E2 29853.793} C_VEL
LIN {X 0,Y 624.901,Z 343.385,A -85,B 0,C 180,E1 29850.579,E2 29850.579} C_VEL
LIN {X 0,Y 624.898,Z 343.39,A -85,B 0,C 180,E1 29847.803,E2 29847.803} C_VEL
LIN {X 0,Y 624.905,Z 343.388,A -85,B 0,C 180,E1 29844.531,E2 29844.531} C_VEL
LIN {X 0,Y 624.896,Z 343.389,A -85,B 0,C 180,E1 29841.739,E2 29841.739} C_VEL
LIN {X 0,Y 624.91,Z 343.387,A -85,B 0,C 180,E1 29838.489,E2 29838.489} C_VEL
LIN {X 0,Y 624.895,Z 343.39,A -85,B 0,C 180,E1 29835.634,E2 29835.634} C_VEL
LIN {X 0,Y 624.917,Z 343.598,A -85,B 0,C 180,E1 29834.076,E2 29834.076} C_VEL
LIN {X 0,Y 633.318,Z 364.488,A -85,B 0,C 180,E1 29831.483,E2 29831.483} C_VEL
LIN {X 0,Y 637.458,Z 375.458,A -85,B 0,C 180,E1 29830.244,E2 29830.244} C_VEL
LIN {X 0,Y 644.114,Z 387.269,A -85,B 0,C 180,E1 29829.57,E2 29829.57} C_VEL
LIN {X 0,Y 648.865,Z 408.283,A -85,B 0,C 180,E1 29828.928,E2 29828.928} C_VEL
LIN {X 0,Y 644.789,Z 676.123,A -85,B 0,C 180,E1 29825.546,E2 29825.546} C_VEL
LIN {X 0,Y 643.359,Z 767.457,A -85,B 0,C 180,E1 29824.388,E2 29824.388} C_VEL
LIN {X 0,Y 642.441,Z 792.729,A -85,B 0,C 180,E1 29823.912,E2 29823.912} C_VEL
LIN {X 0,Y 641.474,Z 812.839,A -85,B 0,C 180,E1 29823.406,E2 29823.406} C_VEL
LIN {X 0,Y 640.273,Z 835.294,A -85,B 0,C 180,E1 29822.706,E2 29822.706} C_VEL
LIN {X 0,Y 638.713,Z 858.184,A -85,B 0,C 180,E1 29821.817,E2 29821.817} C_VEL
LIN {X 0,Y 637.286,Z 878.858,A -85,B 0,C 180,E1 29820.868,E2 29820.868} C_VEL
LIN {X 0,Y 635.566,Z 901.227,A -85,B 0,C 180,E1 29819.655,E2 29819.655} C_VEL
LIN {X 0,Y 634.055,Z 919.856,A -85,B 0,C 180,E1 29818.492,E2 29818.492} C_VEL
LIN {X 0,Y 632.282,Z 941.134,A -85,B 0,C 180,E1 29816.962,E2 29816.962} C_VEL
LIN {X 0,Y 630.831,Z 958.283,A -85,B 0,C 180,E1 29815.539,E2 29815.539} C_VEL
LIN {X 0,Y 629.293,Z 976.747,A -85,B 0,C 180,E1 29813.802,E2 29813.802} C_VEL
LIN {X 0,Y 628.078,Z 991.933,A -85,B 0,C 180,E1 29812.167,E2 29812.167} C_VEL
LIN {X 0,Y 626.909,Z 1007.705,A -85,B 0,C 180,E1 29810.249,E2 29810.249} C_VEL
LIN {X 0,Y 625.997,Z 1021.244,A -85,B 0,C 180,E1 29808.341,E2 29808.341} C_VEL
LIN {X 0,Y 625.286,Z 1033.689,A -85,B 0,C 180,E1 29806.346,E2 29806.346} C_VEL
LIN {X 0,Y 624.723,Z 1044.641,A -85,B 0,C 180,E1 29804.269,E2 29804.269} C_VEL
LIN {X 0,Y 624.367,Z 1053.585,A -85,B 0,C 180,E1 29802.298,E2 29802.298} C_VEL
LIN {X 0,Y 624.106,Z 1061.907,A -85,B 0,C 180,E1 29800.057,E2 29800.057} C_VEL
LIN {X 0,Y 624.01,Z 1067.49,A -85,B 0,C 180,E1 29798.199,E2 29798.199} C_VEL
LIN {X 0,Y 623.94,Z 1072.696,A -85,B 0,C 180,E1 29795.979,E2 29795.979} C_VEL
LIN {X 0,Y 623.907,Z 1076.01,A -85,B 0,C 180,E1 29793.86,E2 29793.86} C_VEL
LIN {X 0,Y 623.904,Z 1077.836,A -85,B 0,C 180,E1 29791.929,E2 29791.929} C_VEL
LIN {X 0,Y 623.895,Z 1078.417,A -85,B 0,C 180,E1 29789.633,E2 29789.633} C_VEL
LIN {X 0,Y 623.91,Z 1077.496,A -85,B 0,C 180,E1 29787.612,E2 29787.612} C_VEL
LIN {X 0,Y 623.919,Z 1075.085,A -85,B 0,C 180,E1 29785.404,E2 29785.404} C_VEL
LIN {X 0,Y 623.939,Z 1071.102,A -85,B 0,C 180,E1 29783.282,E2 29783.282} C_VEL
LIN {X 0,Y 624.014,Z 1066.219,A -85,B 0,C 180,E1 29781.337,E2 29781.337} C_VEL
LIN {X 0,Y 624.206,Z 1058.661,A -85,B 0,C 180,E1 29779.011,E2 29779.011} C_VEL
LIN {X 0,Y 624.476,Z 1050.75,A -85,B 0,C 180,E1 29777.046,E2 29777.046} C_VEL
